LIN {X 0,Y 432.341,Z 420.255,A -85,B 0,C 180,E1 -9394.677,E2 -9394.677} C_VEL
LIN {X 0,Y 432.34,Z 420.258,A -85,B 0,C 180,E1 -9398.15,E2 -9398.15} C_VEL
LIN {X 0,Y 432.366,Z 420.256,A -85,B 0,C 180,E1 -9401.607,E2 -9401.607} C_VEL
LIN {X 0,Y 432.38,Z 420.301,A -85,B 0,C 180,E1 -9402.416,E2 -9402.416} C_VEL
LIN {X 0,Y 432.94,Z 424.326,A -85,B 0,C 180,E1 -9404.417,E2 -9404.417} C_VEL
LIN {X 0,Y 432.411,Z 431.789,A -85,B 0,C 180,E1 -9407.598,E2 -9407.598} C_VEL
LIN {X 0,Y 432.35,Z 439.582,A -85,B 0,C 180,E1 -9410.657,E2 -9410.657} C_VEL
LIN {X 0,Y 432.394,Z 447.543,A -85,B 0,C 180,E1 -9413.611,E2 -9413.611} C_VEL
LIN {X 0,Y 432.393,Z 455.479,A -85,B 0,C 180,E1 -9416.452,E2 -9416.452} C_VEL
LIN {X 0,Y 432.32,Z 464.178,A -85,B 0,C 180,E1 -9419.496,E2 -9419.496} C_VEL
LIN {X 0,Y 432.307,Z 471.048,A -85,B 0,C 180,E1 -9421.871,E2 -9421.871} C_VEL
LIN {X 0,Y 432.174,Z 480.112,A -85,B 0,C 180,E1 -9424.988,E2 -9424.988} C_VEL
LIN {X 0,Y 432.007,Z 490.424,A -85,B 0,C 180,E1 -9428.529,E2 -9428.529} C_VEL
LIN {X 0,Y 431.947,Z 493.135,A -85,B 0,C 180,E1 -9429.462,E2 -9429.462} C_VEL
LIN {X 0,Y 434.775,Z 513.471,A -85,B 0,C 180,E1 -9430.263,E2 -9430.263} C_VEL
LIN {X 0,Y 437.291,Z 527.402,A -85,B 0,C 180,E1 -9430.999,E2 -9430.999} C_VEL
LIN {X 0,Y 437.197,Z 533.625,A -85,B 0,C 180,E1 -9431.331,E2 -9431.331} C_VEL
LIN {X 0,Y 436.147,Z 551.64,A -85,B 0,C 180,E1 -9432.414,E2 -9432.414} C_VEL
LIN {X 0,Y 435.39,Z 563.892,A -85,B 0,C 180,E1 -9433.35,E2 -9433.35} C_VEL
LIN {X 0,Y 434.553,Z 575.091,A -85,B 0,C 180,E1 -9434.403,E2 -9434.403} C_VEL
LIN {X 0,Y 433.711,Z 586.298,A -85,B 0,C 180,E1 -9435.693,E2 -9435.693} C_VEL
LIN {X 0,Y 432.95,Z 596.88,A -85,B 0,C 180,E1 -9437.195,E2 -9437.195} C_VEL
LIN {X 0,Y 432.374,Z 605.824,A -85,B 0,C 180,E1 -9438.752,E2 -9438.752} C_VEL
LIN {X 0,Y 431.951,Z 612.495,A -85,B 0,C 180,E1 -9440.163,E2 -9440.163} C_VEL
LIN {X 0,Y 431.63,Z 618.023,A -85,B 0,C 180,E1 -9441.573,E2 -9441.573} C_VEL
LIN {X 0,Y 431.412,Z 623.802,A -85,B 0,C 180,E1 -9443.452,E2 -9443.452} C_VEL
LIN {X 0,Y 431.277,Z 627.993,A -85,B 0,C 180,E1 -9445.326,E2 -9445.326} C_VEL
LIN {X 0,Y 431.265,Z 630.732,A -85,B 0,C 180,E1 -9447.198,E2 -9447.198} C_VEL
LIN {X 0,Y 431.227,Z 632.093,A -85,B 0,C 180,E1 -9449.066,E2 -9449.066} C_VEL
LIN {X 0,Y 431.227,Z 632.094,A -85,B 0,C 180,E1 -9450.934,E2 -9450.934} C_VEL
LIN {X 0,Y 431.268,Z 630.735,A -85,B 0,C 180,E1 -9452.802,E2 -9452.802} C_VEL
LIN {X 0,Y 431.266,Z 627.997,A -85,B 0,C 180,E1 -9454.674,E2 -9454.674} C_VEL
LIN {X 0,Y 431.407,Z 623.802,A -85,B 0,C 180,E1 -9456.548,E2 -9456.548} C_VEL
LIN {X 0,Y 431.622,Z 618.022,A -85,B 0,C 180,E1 -9458.427,E2 -9458.427} C_VEL
LIN {X 0,Y 431.973,Z 611.488,A -85,B 0,C 180,E1 -9460.073,E2 -9460.073} C_VEL
LIN {X 0,Y 432.528,Z 603.346,A -85,B 0,C 180,E1 -9461.719,E2 -9461.719} C_VEL
LIN {X 0,Y 433.044,Z 594.648,A -85,B 0,C 180,E1 -9463.155,E2 -9463.155} C_VEL
LIN {X 0,Y 433.83,Z 584.413,A -85,B 0,C 180,E1 -9464.543,E2 -9464.543} C_VEL
LIN {X 0,Y 434.781,Z 571.943,A -85,B 0,C 180,E1 -9465.95,E2 -9465.95} C_VEL
LIN {X 0,Y 435.848,Z 559.24,A -85,B 0,C 180,E1 -9467.114,E2 -9467.114} C_VEL
LIN {X 0,Y 436.767,Z 546.427,A -85,B 0,C 180,E1 -9468.06,E2 -9468.06} C_VEL
LIN {X 0,Y 437.539,Z 533.501,A -85,B 0,C 180,E1 -9468.82,E2 -9468.82} C_VEL
LIN {X 0,Y 437.702,Z 528.722,A -85,B 0,C 180,E1 -9469.057,E2 -9469.057} C_VEL
LIN {X 0,Y 435.149,Z 514.725,A -85,B 0,C 180,E1 -9469.765,E2 -9469.765} C_VEL
LIN {X 0,Y 432.262,Z 499.953,A -85,B 0,C 180,E1 -9470.339,E2 -9470.339} C_VEL
LIN {X 0,Y 431.957,Z 497.779,A -85,B 0,C 180,E1 -9470.426,E2 -9470.426} C_VEL
LIN {X 0,Y 432.221,Z 489.918,A -85,B 0,C 180,E1 -9473.477,E2 -9473.477} C_VEL
LIN {X 0,Y 432.485,Z 481.872,A -85,B 0,C 180,E1 -9476.65,E2 -9476.65} C_VEL
LIN {X 0,Y 432.838,Z 474.315,A -85,B 0,C 180,E1 -9479.685,E2 -9479.685} C_VEL
LIN {X 0,Y 433.175,Z 466.427,A -85,B 0,C 180,E1 -9482.924,E2 -9482.924} C_VEL
LIN {X 0,Y 433.444,Z 459.515,A -85,B 0,C 180,E1 -9485.834,E2 -9485.834} C_VEL
LIN {X 0,Y 433.752,Z 451.761,A -85,B 0,C 180,E1 -9489.191,E2 -9489.191} C_VEL
LIN {X 0,Y 434.086,Z 445.759,A -85,B 0,C 180,E1 -9491.862,E2 -9491.862} C_VEL
LIN {X 0,Y 434.542,Z 438.136,A -85,B 0,C 180,E1 -9495.368,E2 -9495.368} C_VEL
LIN {X 0,Y 434.616,Z 434.256,A -85,B 0,C 180,E1 -9497.222,E2 -9497.222} C_VEL
LIN {X 0,Y 433.981,Z 429.502,A -85,B 0,C 180,E1 -9499.626,E2 -9499.626} C_VEL
LIN {X 0,Y 432.949,Z 423.719,A -85,B 0,C 180,E1 -9502.694,E2 -9502.694} C_VEL
LIN {X 0,Y 432.371,Z 420.252,A -85,B 0,C 180,E1 -9504.717,E2 -9504.717} C_VEL
LIN {X 0,Y 432.326,Z 420.259,A -85,B 0,C 180,E1 -9507.707,E2 -9507.707} C_VEL
LIN {X 0,Y 432.344,Z 420.257,A -85,B 0,C 180,E1 -9510.813,E2 -9510.813} C_VEL
LIN {X 0,Y 432.366,Z 420.243,A -85,B 0,C 180,E1 -9513.968,E2 -9513.968} C_VEL
LIN {X 0,Y 432.321,Z 420.259,A -85,B 0,C 180,E1 -9517.036,E2 -9517.036} C_VEL
LIN {X 0,Y 432.389,Z 420.245,A -85,B 0,C 180,E1 -9520.515,E2 -9520.515} C_VEL
LIN {X 0,Y 432.433,Z 420.239,A -85,B 0,C 180,E1 -9523.961,E2 -9523.961} C_VEL
LIN {X 0,Y 432.461,Z 420.242,A -85,B 0,C 180,E1 -9527.804,E2 -9527.804} C_VEL
LIN {X 0,Y 432.466,Z 420.232,A -85,B 0,C 180,E1 -9531.59,E2 -9531.59} C_VEL
LIN {X 0,Y 432.598,Z 420.224,A -85,B 0,C 180,E1 -9534.406,E2 -9534.406} C_VEL
LIN {X 0,Y 432.606,Z 420.216,A -85,B 0,C 180,E1 -9538.138,E2 -9538.138} C_VEL
LIN {X 0,Y 432.736,Z 420.21,A -85,B 0,C 180,E1 -9540,E2 -9540} C_VEL
LIN {X 0,Y 432.594,Z 420.215,A -85,B 0,C 180,E1 -9542.794,E2 -9542.794} C_VEL
LIN {X 0,Y 432.575,Z 420.226,A -85,B 0,C 180,E1 -9546.53,E2 -9546.53} C_VEL
LIN {X 0,Y 432.445,Z 420.238,A -85,B 0,C 180,E1 -9549.353,E2 -9549.353} C_VEL
LIN {X 0,Y 432.433,Z 420.241,A -85,B 0,C 180,E1 -9552.804,E2 -9552.804} C_VEL
LIN {X 0,Y 432.415,Z 420.251,A -85,B 0,C 180,E1 -9556.479,E2 -9556.479} C_VEL
LIN {X 0,Y 432.342,Z 420.257,A -85,B 0,C 180,E1 -9559.96,E2 -9559.96} C_VEL
LIN {X 0,Y 432.319,Z 420.253,A -85,B 0,C 180,E1 -9562.964,E2 -9562.964} C_VEL
LIN {X 0,Y 432.363,Z 420.25,A -85,B 0,C 180,E1 -9566.033,E2 -9566.033} C_VEL
LIN {X 0,Y 432.345,Z 420.254,A -85,B 0,C 180,E1 -9569.187,E2 -9569.187} C_VEL
LIN {X 0,Y 432.325,Z 420.258,A -85,B 0,C 180,E1 -9572.443,E2 -9572.443} C_VEL
LIN {X 0,Y 432.346,Z 420.254,A -85,B 0,C 180,E1 -9575.632,E2 -9575.632} C_VEL
LIN {X 0,Y 432.352,Z 420.256,A -85,B 0,C 180,E1 -9579.343,E2 -9579.343} C_VEL
LIN {X 0,Y 432.337,Z 420.258,A -85,B 0,C 180,E1 -9581.797,E2 -9581.797} C_VEL
LIN {X 0,Y 432.343,Z 420.256,A -85,B 0,C 180,E1 -9584.346,E2 -9584.346} C_VEL
LIN {X 0,Y 432.367,Z 420.365,A -85,B 0,C 180,E1 -9587.395,E2 -9587.395} C_VEL
LIN {X 0,Y 434.001,Z 428.984,A -85,B 0,C 180,E1 -9590.244,E2 -9590.244} C_VEL
LIN {X 0,Y 434.458,Z 432.86,A -85,B 0,C 180,E1 -9591.529,E2 -9591.529} C_VEL
LIN {X 0,Y 434.028,Z 441.711,A -85,B 0,C 180,E1 -9594.343,E2 -9594.343} C_VEL
LIN {X 0,Y 433.727,Z 452.025,A -85,B 0,C 180,E1 -9597.675,E2 -9597.675} C_VEL
LIN {X 0,Y 433.428,Z 462.73,A -85,B 0,C 180,E1 -9601.117,E2 -9601.117} C_VEL
LIN {X 0,Y 433.024,Z 473.572,A -85,B 0,C 180,E1 -9604.526,E2 -9604.526} C_VEL
LIN {X 0,Y 432.751,Z 484.213,A -85,B 0,C 180,E1 -9607.774,E2 -9607.774} C_VEL
LIN {X 0,Y 432.631,Z 491.462,A -85,B 0,C 180,E1 -9609.853,E2 -9609.853} C_VEL
LIN {X 0,Y 436.02,Z 506.623,A -85,B 0,C 180,E1 -9610.365,E2 -9610.365} C_VEL
LIN {X 0,Y 438.052,Z 518.136,A -85,B 0,C 180,E1 -9610.87,E2 -9610.87} C_VEL
LIN {X 0,Y 437.448,Z 530.781,A -85,B 0,C 180,E1 -9611.453,E2 -9611.453} C_VEL
LIN {X 0,Y 436.825,Z 543.155,A -85,B 0,C 180,E1 -9612.2,E2 -9612.2} C_VEL
LIN {X 0,Y 435.927,Z 555.472,A -85,B 0,C 180,E1 -9613.13,E2 -9613.13} C_VEL
LIN {X 0,Y 435.057,Z 566.744,A -85,B 0,C 180,E1 -9614.181,E2 -9614.181} C_VEL
LIN {X 0,Y 434.187,Z 578.069,A -85,B 0,C 180,E1 -9615.47,E2 -9615.47} C_VEL
LIN {X 0,Y 433.304,Z 588.216,A -85,B 0,C 180,E1 -9616.875,E2 -9616.875} C_VEL
LIN {X 0,Y 432.77,Z 596.592,A -85,B 0,C 180,E1 -9618.288,E2 -9618.288} C_VEL
LIN {X 0,Y 432.142,Z 604.593,A -85,B 0,C 180,E1 -9619.931,E2 -9619.931} C_VEL
LIN {X 0,Y 431.988,Z 606.62,A -85,B 0,C 180,E1 -9620.414,E2 -9620.414} C_VEL
LIN {X 0,Y 431.169,Z 609.388,A -85,B 0,C 180,E1 -9621.099,E2 -9621.099} C_VEL
LIN {X 0,Y 428.07,Z 613.464,A -85,B 0,C 180,E1 -9622.233,E2 -9622.233} C_VEL
LIN {X 0,Y 425.022,Z 616.961,A -85,B 0,C 180,E1 -9623.416,E2 -9623.416} C_VEL
LIN {X 0,Y 424.294,Z 618.757,A -85,B 0,C 180,E1 -9624.169,E2 -9624.169} C_VEL
LIN {X 0,Y 424.201,Z 620.94,A -85,B 0,C 180,E1 -9625.248,E2 -9625.248} C_VEL
LIN {X 0,Y 424.122,Z 623.658,A -85,B 0,C 180,E1 -9627.151,E2 -9627.151} C_VEL
LIN {X 0,Y 424.067,Z 625.023,A -85,B 0,C 180,E1 -9629.05,E2 -9629.05} C_VEL
LIN {X 0,Y 424.067,Z 625.061,A -85,B 0,C 180,E1 -9630.95,E2 -9630.95} C_VEL
LIN {X 0,Y 424.121,Z 623.762,A -85,B 0,C 180,E1 -9632.849,E2 -9632.849} C_VEL
LIN {X 0,Y 424.201,Z 621.106,A -85,B 0,C 180,E1 -9634.752,E2 -9634.752} C_VEL
LIN {X 0,Y 424.354,Z 617.026,A -85,B 0,C 180,E1 -9636.657,E2 -9636.657} C_VEL
LIN {X 0,Y 424.63,Z 611.396,A -85,B 0,C 180,E1 -9638.567,E2 -9638.567} C_VEL
LIN {X 0,Y 425.001,Z 606.024,A -85,B 0,C 180,E1 -9639.999,E2 -9639.999} C_VEL
LIN {X 0,Y 425.655,Z 598.336,A -85,B 0,C 180,E1 -9641.669,E2 -9641.669} C_VEL
LIN {X 0,Y 426.236,Z 590.302,A -85,B 0,C 180,E1 -9643.104,E2 -9643.104} C_VEL
LIN {X 0,Y 427.052,Z 580.624,A -85,B 0,C 180,E1 -9644.535,E2 -9644.535} C_VEL
LIN {X 0,Y 427.941,Z 569.882,A -85,B 0,C 180,E1 -9645.845,E2 -9645.845} C_VEL
LIN {X 0,Y 428.948,Z 557.958,A -85,B 0,C 180,E1 -9647.03,E2 -9647.03} C_VEL
LIN {X 0,Y 429.832,Z 546.206,A -85,B 0,C 180,E1 -9647.976,E2 -9647.976} C_VEL
LIN {X 0,Y 430.684,Z 532.74,A -85,B 0,C 180,E1 -9648.833,E2 -9648.833} C_VEL
LIN {X 0,Y 431.257,Z 518.562,A -85,B 0,C 180,E1 -9649.52,E2 -9649.52} C_VEL
LIN {X 0,Y 428.609,Z 504.1,A -85,B 0,C 180,E1 -9650.158,E2 -9650.158} C_VEL
LIN {X 0,Y 425.583,Z 491.211,A -85,B 0,C 180,E1 -9650.611,E2 -9650.611} C_VEL
LIN {X 0,Y 425.832,Z 482.093,A -85,B 0,C 180,E1 -9653.335,E2 -9653.335} C_VEL
LIN {X 0,Y 426.12,Z 472.049,A -85,B 0,C 180,E1 -9656.443,E2 -9656.443} C_VEL
LIN {X 0,Y 426.493,Z 462.064,A -85,B 0,C 180,E1 -9659.627,E2 -9659.627} C_VEL
LIN {X 0,Y 426.83,Z 451.984,A -85,B 0,C 180,E1 -9662.913,E2 -9662.913} C_VEL
LIN {X 0,Y 427.166,Z 441.511,A -85,B 0,C 180,E1 -9666.32,E2 -9666.32} C_VEL
LIN {X 0,Y 427.515,Z 434.261,A -85,B 0,C 180,E1 -9668.659,E2 -9668.659} C_VEL
LIN {X 0,Y 426.638,Z 428.084,A -85,B 0,C 180,E1 -9670.733,E2 -9670.733} C_VEL
LIN {X 0,Y 425.271,Z 421.14,A -85,B 0,C 180,E1 -9673.102,E2 -9673.102} C_VEL
LIN {X 0,Y 425.271,Z 421.14,A -85,B 0,C 180,E1 -9676.045,E2 -9676.045} C_VEL
LIN {X 0,Y 425.277,Z 421.141,A -85,B 0,C 180,E1 -9678.622,E2 -9678.622} C_VEL
LIN {X 0,Y 425.311,Z 421.136,A -85,B 0,C 180,E1 -9681.102,E2 -9681.102} C_VEL
LIN {X 0,Y 425.302,Z 421.134,A -85,B 0,C 180,E1 -9684.664,E2 -9684.664} C_VEL
LIN {X 0,Y 425.268,Z 421.138,A -85,B 0,C 180,E1 -9688.073,E2 -9688.073} C_VEL
LIN {X 0,Y 425.34,Z 421.13,A -85,B 0,C 180,E1 -9691.368,E2 -9691.368} C_VEL
LIN {X 0,Y 425.298,Z 421.133,A -85,B 0,C 180,E1 -9694.555,E2 -9694.555} C_VEL
LIN {X 0,Y 425.311,Z 421.132,A -85,B 0,C 180,E1 -9697.662,E2 -9697.662} C_VEL
LIN {X 0,Y 430.712,Z 437.499,A -85,B 0,C 180,E1 -9698.779,E2 -9698.779} C_VEL
LIN {X 0,Y 431.814,Z 441.37,A -85,B 0,C 180,E1 -9699.073,E2 -9699.073} C_VEL
LIN {X 0,Y 431.099,Z 454.659,A -85,B 0,C 180,E1 -9699.98,E2 -9699.98} C_VEL
LIN {X 0,Y 430.149,Z 467.57,A -85,B 0,C 180,E1 -9701.048,E2 -9701.048} C_VEL
LIN {X 0,Y 429.193,Z 479.566,A -85,B 0,C 180,E1 -9702.243,E2 -9702.243} C_VEL
LIN {X 0,Y 428.33,Z 490.646,A -85,B 0,C 180,E1 -9703.558,E2 -9703.558} C_VEL
LIN {X 0,Y 427.497,Z 500.849,A -85,B 0,C 180,E1 -9704.993,E2 -9704.993} C_VEL
LIN {X 0,Y 426.638,Z 510.775,A -85,B 0,C 180,E1 -9706.666,E2 -9706.666} C_VEL
LIN {X 0,Y 426.05,Z 519.022,A -85,B 0,C 180,E1 -9708.342,E2 -9708.342} C_VEL
LIN {X 0,Y 425.544,Z 525.822,A -85,B 0,C 180,E1 -9710.014,E2 -9710.014} C_VEL
LIN {X 0,Y 425.121,Z 532.087,A -85,B 0,C 180,E1 -9711.922,E2 -9711.922} C_VEL
LIN {X 0,Y 424.842,Z 536.907,A -85,B 0,C 180,E1 -9713.827,E2 -9713.827} C_VEL
LIN {X 0,Y 424.748,Z 539.643,A -85,B 0,C 180,E1 -9715.254,E2 -9715.254} C_VEL
LIN {X 0,Y 424.556,Z 542.251,A -85,B 0,C 180,E1 -9717.153,E2 -9717.153} C_VEL
LIN {X 0,Y 424.378,Z 543.678,A -85,B 0,C 180,E1 -9719.051,E2 -9719.051} C_VEL
LIN {X 0,Y 424.396,Z 543.894,A -85,B 0,C 180,E1 -9720.949,E2 -9720.949} C_VEL
LIN {X 0,Y 424.574,Z 542.936,A -85,B 0,C 180,E1 -9722.846,E2 -9722.846} C_VEL
LIN {X 0,Y 424.928,Z 540.794,A -85,B 0,C 180,E1 -9724.744,E2 -9724.744} C_VEL
LIN {X 0,Y 425.099,Z 537.458,A -85,B 0,C 180,E1 -9726.646,E2 -9726.646} C_VEL
LIN {X 0,Y 425.51,Z 532.778,A -85,B 0,C 180,E1 -9728.549,E2 -9728.549} C_VEL
LIN {X 0,Y 425.878,Z 526.647,A -85,B 0,C 180,E1 -9730.459,E2 -9730.459} C_VEL
LIN {X 0,Y 426.612,Z 518.868,A -85,B 0,C 180,E1 -9732.366,E2 -9732.366} C_VEL
LIN {X 0,Y 427.378,Z 510.571,A -85,B 0,C 180,E1 -9734.017,E2 -9734.017} C_VEL
LIN {X 0,Y 428.181,Z 501.807,A -85,B 0,C 180,E1 -9735.469,E2 -9735.469} C_VEL
LIN {X 0,Y 429.024,Z 491.512,A -85,B 0,C 180,E1 -9736.904,E2 -9736.904} C_VEL
LIN {X 0,Y 430.029,Z 479.806,A -85,B 0,C 180,E1 -9738.264,E2 -9738.264} C_VEL
LIN {X 0,Y 431.049,Z 467.92,A -85,B 0,C 180,E1 -9739.402,E2 -9739.402} C_VEL
LIN {X 0,Y 431.824,Z 456.017,A -85,B 0,C 180,E1 -9740.358,E2 -9740.358} C_VEL
LIN {X 0,Y 432.604,Z 441.693,A -85,B 0,C 180,E1 -9741.291,E2 -9741.291} C_VEL
LIN {X 0,Y 429.046,Z 430.815,A -85,B 0,C 180,E1 -9742.133,E2 -9742.133} C_VEL
LIN {X 0,Y 425.334,Z 421.52,A -85,B 0,C 180,E1 -9742.806,E2 -9742.806} C_VEL
LIN {X 0,Y 425.273,Z 421.137,A -85,B 0,C 180,E1 -9742.853,E2 -9742.853} C_VEL
LIN {X 0,Y 425.292,Z 421.139,A -85,B 0,C 180,E1 -9745.445,E2 -9745.445} C_VEL
LIN {X 0,Y 425.351,Z 421.132,A -85,B 0,C 180,E1 -9747.558,E2 -9747.558} C_VEL
LIN {X 0,Y 425.289,Z 421.133,A -85,B 0,C 180,E1 -9750.816,E2 -9750.816} C_VEL
LIN {X 0,Y 425.312,Z 421.132,A -85,B 0,C 180,E1 -9754.288,E2 -9754.288} C_VEL
LIN {X 0,Y 425.281,Z 421.138,A -85,B 0,C 180,E1 -9757.694,E2 -9757.694} C_VEL
LIN {X 0,Y 425.286,Z 421.136,A -85,B 0,C 180,E1 -9760.521,E2 -9760.521} C_VEL
LIN {X 0,Y 425.371,Z 421.276,A -85,B 0,C 180,E1 -9762.165,E2 -9762.165} C_VEL
LIN {X 0,Y 425.885,Z 424.541,A -85,B 0,C 180,E1 -9763.875,E2 -9763.875} C_VEL
LIN {X 0,Y 425.733,Z 428.375,A -85,B 0,C 180,E1 -9765.647,E2 -9765.647} C_VEL
LIN {X 0,Y 425.336,Z 438.536,A -85,B 0,C 180,E1 -9769.878,E2 -9769.878} C_VEL
LIN {X 0,Y 425.342,Z 446.633,A -85,B 0,C 180,E1 -9772.992,E2 -9772.992} C_VEL
LIN {X 0,Y 425.338,Z 454.302,A -85,B 0,C 180,E1 -9775.82,E2 -9775.82} C_VEL
LIN {X 0,Y 425.262,Z 463.858,A -85,B 0,C 180,E1 -9779.246,E2 -9779.246} C_VEL
LIN {X 0,Y 425.207,Z 471.366,A -85,B 0,C 180,E1 -9781.897,E2 -9781.897} C_VEL
LIN {X 0,Y 425.091,Z 480.314,A -85,B 0,C 180,E1 -9785.03,E2 -9785.03} C_VEL
LIN {X 0,Y 424.905,Z 490.694,A -85,B 0,C 180,E1 -9788.661,E2 -9788.661} C_VEL
LIN {X 0,Y 424.871,Z 492.011,A -85,B 0,C 180,E1 -9789.057,E2 -9789.057} C_VEL
LIN {X 0,Y 427.326,Z 508.383,A -85,B 0,C 180,E1 -9789.704,E2 -9789.704} C_VEL
LIN {X 0,Y 428.466,Z 517.12,A -85,B 0,C 180,E1 -9790.121,E2 -9790.121} C_VEL
LIN {X 0,Y 430.611,Z 530.032,A -85,B 0,C 180,E1 -9790.867,E2 -9790.867} C_VEL
LIN {X 0,Y 429.581,Z 548.076,A -85,B 0,C 180,E1 -9791.89,E2 -9791.89} C_VEL
LIN {X 0,Y 428.744,Z 560.999,A -85,B 0,C 180,E1 -9792.839,E2 -9792.839} C_VEL
LIN {X 0,Y 427.835,Z 572.697,A -85,B 0,C 180,E1 -9793.907,E2 -9793.907} C_VEL
LIN {X 0,Y 427.115,Z 582.402,A -85,B 0,C 180,E1 -9794.98,E2 -9794.98} C_VEL
LIN {X 0,Y 426.289,Z 593.119,A -85,B 0,C 180,E1 -9796.412,E2 -9796.412} C_VEL
LIN {X 0,Y 425.667,Z 601.943,A -85,B 0,C 180,E1 -9797.848,E2 -9797.848} C_VEL
LIN {X 0,Y 424.993,Z 610.376,A -85,B 0,C 180,E1 -9799.519,E2 -9799.519} C_VEL
LIN {X 0,Y 424.679,Z 616.242,A -85,B 0,C 180,E1 -9800.955,E2 -9800.955} C_VEL
LIN {X 0,Y 424.346,Z 622.488,A -85,B 0,C 180,E1 -9802.865,E2 -9802.865} C_VEL
LIN {X 0,Y 424.283,Z 626.029,A -85,B 0,C 180,E1 -9804.296,E2 -9804.296} C_VEL
LIN {X 0,Y 424.196,Z 629.481,A -85,B 0,C 180,E1 -9806.2,E2 -9806.2} C_VEL
LIN {X 0,Y 424.196,Z 631.525,A -85,B 0,C 180,E1 -9808.101,E2 -9808.101} C_VEL
LIN {X 0,Y 424.116,Z 632.205,A -85,B 0,C 180,E1 -9810,E2 -9810} C_VEL
LIN {X 0,Y 424.196,Z 631.526,A -85,B 0,C 180,E1 -9811.899,E2 -9811.899} C_VEL
LIN {X 0,Y 424.193,Z 629.485,A -85,B 0,C 180,E1 -9813.8,E2 -9813.8} C_VEL
LIN {X 0,Y 424.254,Z 626.032,A -85,B 0,C 180,E1 -9815.704,E2 -9815.704} C_VEL
LIN {X 0,Y 424.364,Z 621.062,A -85,B 0,C 180,E1 -9817.614,E2 -9817.614} C_VEL
LIN {X 0,Y 424.642,Z 616.24,A -85,B 0,C 180,E1 -9819.046,E2 -9819.046} C_VEL
LIN {X 0,Y 425.086,Z 609.261,A -85,B 0,C 180,E1 -9820.719,E2 -9820.719} C_VEL
LIN {X 0,Y 425.725,Z 600.588,A -85,B 0,C 180,E1 -9822.393,E2 -9822.393} C_VEL
LIN {X 0,Y 426.389,Z 591.492,A -85,B 0,C 180,E1 -9823.827,E2 -9823.827} C_VEL
LIN {X 0,Y 427.107,Z 582.401,A -85,B 0,C 180,E1 -9825.021,E2 -9825.021} C_VEL
LIN {X 0,Y 427.9,Z 571.524,A -85,B 0,C 180,E1 -9826.213,E2 -9826.213} C_VEL
LIN {X 0,Y 429.087,Z 557.222,A -85,B 0,C 180,E1 -9827.516,E2 -9827.516} C_VEL
LIN {X 0,Y 430.106,Z 543.368,A -85,B 0,C 180,E1 -9828.525,E2 -9828.525} C_VEL
LIN {X 0,Y 430.924,Z 530.38,A -85,B 0,C 180,E1 -9829.265,E2 -9829.265} C_VEL
LIN {X 0,Y 428.616,Z 516.863,A -85,B 0,C 180,E1 -9829.991,E2 -9829.991} C_VEL
LIN {X 0,Y 425.763,Z 501.841,A -85,B 0,C 180,E1 -9830.621,E2 -9830.621} C_VEL
LIN {X 0,Y 424.911,Z 497.198,A -85,B 0,C 180,E1 -9830.78,E2 -9830.78} C_VEL
LIN {X 0,Y 425.189,Z 489.344,A -85,B 0,C 180,E1 -9833.889,E2 -9833.889} C_VEL
LIN {X 0,Y 425.431,Z 481.945,A -85,B 0,C 180,E1 -9836.866,E2 -9836.866} C_VEL
LIN {X 0,Y 425.787,Z 475.043,A -85,B 0,C 180,E1 -9839.681,E2 -9839.681} C_VEL
LIN {X 0,Y 426.124,Z 467.15,A -85,B 0,C 180,E1 -9842.974,E2 -9842.974} C_VEL
LIN {X 0,Y 426.438,Z 459.748,A -85,B 0,C 180,E1 -9846.142,E2 -9846.142} C_VEL
LIN {X 0,Y 426.743,Z 452.616,A -85,B 0,C 180,E1 -9849.282,E2 -9849.282} C_VEL
LIN {X 0,Y 427.107,Z 446.106,A -85,B 0,C 180,E1 -9852.229,E2 -9852.229} C_VEL
LIN {X 0,Y 427.573,Z 438.808,A -85,B 0,C 180,E1 -9855.643,E2 -9855.643} C_VEL
LIN {X 0,Y 427.549,Z 434.583,A -85,B 0,C 180,E1 -9857.706,E2 -9857.706} C_VEL
LIN {X 0,Y 426.906,Z 430.032,A -85,B 0,C 180,E1 -9860.056,E2 -9860.056} C_VEL
LIN {X 0,Y 425.74,Z 423.598,A -85,B 0,C 180,E1 -9863.539,E2 -9863.539} C_VEL
LIN {X 0,Y 425.319,Z 421.13,A -85,B 0,C 180,E1 -9864.95,E2 -9864.95} C_VEL
LIN {X 0,Y 425.266,Z 421.139,A -85,B 0,C 180,E1 -9868.073,E2 -9868.073} C_VEL
LIN {X 0,Y 425.333,Z 421.133,A -85,B 0,C 180,E1 -9871.368,E2 -9871.368} C_VEL
LIN {X 0,Y 425.297,Z 421.126,A -85,B 0,C 180,E1 -9874.555,E2 -9874.555} C_VEL
LIN {X 0,Y 425.289,Z 421.132,A -85,B 0,C 180,E1 -9877.661,E2 -9877.661} C_VEL
LIN {X 0,Y 425.364,Z 421.122,A -85,B 0,C 180,E1 -9880.704,E2 -9880.704} C_VEL
LIN {X 0,Y 425.39,Z 421.117,A -85,B 0,C 180,E1 -9883.688,E2 -9883.688} C_VEL
LIN {X 0,Y 425.414,Z 421.118,A -85,B 0,C 180,E1 -9887.598,E2 -9887.598} C_VEL
LIN {X 0,Y 425.41,Z 421.109,A -85,B 0,C 180,E1 -9891.449,E2 -9891.449} C_VEL
LIN {X 0,Y 425.554,Z 421.102,A -85,B 0,C 180,E1 -9894.313,E2 -9894.313} C_VEL
LIN {X 0,Y 425.575,Z 421.091,A -85,B 0,C 180,E1 -9898.107,E2 -9898.107} C_VEL
LIN {X 0,Y 425.705,Z 421.086,A -85,B 0,C 180,E1 -9900,E2 -9900} C_VEL
LIN {X 0,Y 425.547,Z 421.092,A -85,B 0,C 180,E1 -9902.84,E2 -9902.84} C_VEL
LIN {X 0,Y 425.533,Z 421.102,A -85,B 0,C 180,E1 -9906.639,E2 -9906.639} C_VEL
LIN {X 0,Y 425.403,Z 421.117,A -85,B 0,C 180,E1 -9909.509,E2 -9909.509} C_VEL
LIN {X 0,Y 425.395,Z 421.117,A -85,B 0,C 180,E1 -9912.904,E2 -9912.904} C_VEL
LIN {X 0,Y 425.364,Z 421.128,A -85,B 0,C 180,E1 -9916.605,E2 -9916.605} C_VEL
LIN {X 0,Y 425.331,Z 421.127,A -85,B 0,C 180,E1 -9919.636,E2 -9919.636} C_VEL
LIN {X 0,Y 425.289,Z 421.132,A -85,B 0,C 180,E1 -9922.339,E2 -9922.339} C_VEL
LIN {X 0,Y 425.293,Z 421.136,A -85,B 0,C 180,E1 -9925.446,E2 -9925.446} C_VEL
LIN {X 0,Y 425.351,Z 421.127,A -85,B 0,C 180,E1 -9927.558,E2 -9927.558} C_VEL
LIN {X 0,Y 425.29,Z 421.133,A -85,B 0,C 180,E1 -9930.816,E2 -9930.816} C_VEL
LIN {X 0,Y 425.313,Z 421.133,A -85,B 0,C 180,E1 -9934.288,E2 -9934.288} C_VEL
LIN {X 0,Y 425.281,Z 421.135,A -85,B 0,C 180,E1 -9937.694,E2 -9937.694} C_VEL
LIN {X 0,Y 425.284,Z 421.138,A -85,B 0,C 180,E1 -9940.521,E2 -9940.521} C_VEL
LIN {X 0,Y 425.266,Z 421.139,A -85,B 0,C 180,E1 -9943.352,E2 -9943.352} C_VEL
LIN {X 0,Y 425.262,Z 421.142,A -85,B 0,C 180,E1 -9946.044,E2 -9946.044} C_VEL
LIN {X 0,Y 425.301,Z 421.276,A -85,B 0,C 180,E1 -9947.085,E2 -9947.085} C_VEL
LIN {X 0,Y 427.023,Z 430.139,A -85,B 0,C 180,E1 -9950.069,E2 -9950.069} C_VEL
LIN {X 0,Y 427.494,Z 435.311,A -85,B 0,C 180,E1 -9951.782,E2 -9951.782} C_VEL
LIN {X 0,Y 427.03,Z 444.714,A -85,B 0,C 180,E1 -9954.829,E2 -9954.829} C_VEL
LIN {X 0,Y 426.681,Z 455.063,A -85,B 0,C 180,E1 -9958.191,E2 -9958.191} C_VEL
LIN {X 0,Y 426.378,Z 465.095,A -85,B 0,C 180,E1 -9961.445,E2 -9961.445} C_VEL
LIN {X 0,Y 426.029,Z 475.079,A -85,B 0,C 180,E1 -9964.602,E2 -9964.602} C_VEL
LIN {X 0,Y 425.754,Z 485.137,A -85,B 0,C 180,E1 -9967.687,E2 -9967.687} C_VEL
LIN {X 0,Y 425.619,Z 491.234,A -85,B 0,C 180,E1 -9969.49,E2 -9969.49} C_VEL
LIN {X 0,Y 429.342,Z 507.939,A -85,B 0,C 180,E1 -9970.086,E2 -9970.086} C_VEL
LIN {X 0,Y 431.299,Z 519.458,A -85,B 0,C 180,E1 -9970.614,E2 -9970.614} C_VEL
LIN {X 0,Y 430.646,Z 532.803,A -85,B 0,C 180,E1 -9971.262,E2 -9971.262} C_VEL
LIN {X 0,Y 429.799,Z 546.611,A -85,B 0,C 180,E1 -9972.146,E2 -9972.146} C_VEL
LIN {X 0,Y 428.947,Z 558.279,A -85,B 0,C 180,E1 -9973.093,E2 -9973.093} C_VEL
LIN {X 0,Y 428.123,Z 567.942,A -85,B 0,C 180,E1 -9974.04,E2 -9974.04} C_VEL
LIN {X 0,Y 427.3,Z 578.124,A -85,B 0,C 180,E1 -9975.23,E2 -9975.23} C_VEL
LIN {X 0,Y 426.349,Z 588.272,A -85,B 0,C 180,E1 -9976.657,E2 -9976.657} C_VEL
LIN {X 0,Y 425.797,Z 596.649,A -85,B 0,C 180,E1 -9978.093,E2 -9978.093} C_VEL
LIN {X 0,Y 425.122,Z 604.651,A -85,B 0,C 180,E1 -9979.763,E2 -9979.763} C_VEL
LIN {X 0,Y 424.646,Z 611.088,A -85,B 0,C 180,E1 -9981.434,E2 -9981.434} C_VEL
LIN {X 0,Y 424.354,Z 616.79,A -85,B 0,C 180,E1 -9983.343,E2 -9983.343} C_VEL
LIN {X 0,Y 424.294,Z 618.757,A -85,B 0,C 180,E1 -9984.169,E2 -9984.169} C_VEL
LIN {X 0,Y 423.597,Z 620.409,A -85,B 0,C 180,E1 -9984.929,E2 -9984.929} C_VEL
LIN {X 0,Y 420.693,Z 622.599,A -85,B 0,C 180,E1 -9986.179,E2 -9986.179} C_VEL
LIN {X 0,Y 418.227,Z 623.856,A -85,B 0,C 180,E1 -9987.202,E2 -9987.202} C_VEL
LIN {X 0,Y 417.136,Z 624.512,A -85,B 0,C 180,E1 -9987.998,E2 -9987.998} C_VEL
LIN {X 0,Y 417.029,Z 624.672,A -85,B 0,C 180,E1 -9988.269,E2 -9988.269} C_VEL
LIN {X 0,Y 416.982,Z 625.267,A -85,B 0,C 180,E1 -9990,E2 -9990} C_VEL
LIN {X 0,Y 417.051,Z 624.638,A -85,B 0,C 180,E1 -9991.931,E2 -9991.931} C_VEL
LIN {X 0,Y 417.013,Z 622.664,A -85,B 0,C 180,E1 -9993.865,E2 -9993.865} C_VEL
LIN {X 0,Y 417.198,Z 619.307,A -85,B 0,C 180,E1 -9995.801,E2 -9995.801} C_VEL
LIN {X 0,Y 417.391,Z 614.471,A -85,B 0,C 180,E1 -9997.741,E2 -9997.741} C_VEL
LIN {X 0,Y 417.838,Z 608.001,A -85,B 0,C 180,E1 -9999.683,E2 -9999.683} C_VEL
LIN {X 0,Y 418.389,Z 600.791,A -85,B 0,C 180,E1 -10001.383,E2 -10001.383} C_VEL
LIN {X 0,Y 419.207,Z 592.022,A -85,B 0,C 180,E1 -10003.046,E2 -10003.046} C_VEL
LIN {X 0,Y 420.002,Z 582.419,A -85,B 0,C 180,E1 -10004.537,E2 -10004.537} C_VEL
LIN {X 0,Y 420.944,Z 572.019,A -85,B 0,C 180,E1 -10005.866,E2 -10005.866} C_VEL
LIN {X 0,Y 421.914,Z 560.542,A -85,B 0,C 180,E1 -10007.073,E2 -10007.073} C_VEL
LIN {X 0,Y 422.943,Z 547.824,A -85,B 0,C 180,E1 -10008.154,E2 -10008.154} C_VEL
LIN {X 0,Y 423.817,Z 535.216,A -85,B 0,C 180,E1 -10009.004,E2 -10009.004} C_VEL
LIN {X 0,Y 424.538,Z 521.839,A -85,B 0,C 180,E1 -10009.699,E2 -10009.699} C_VEL
LIN {X 0,Y 424.315,Z 518.305,A -85,B 0,C 180,E1 -10009.864,E2 -10009.864} C_VEL
LIN {X 0,Y 421.771,Z 504.624,A -85,B 0,C 180,E1 -10010.483,E2 -10010.483} C_VEL
LIN {X 0,Y 418.599,Z 491.165,A -85,B 0,C 180,E1 -10010.983,E2 -10010.983} C_VEL
LIN {X 0,Y 418.843,Z 482.005,A -85,B 0,C 180,E1 -10013.748,E2 -10013.748} C_VEL
LIN {X 0,Y 419.178,Z 471.873,A -85,B 0,C 180,E1 -10016.916,E2 -10016.916} C_VEL
LIN {X 0,Y 419.531,Z 461.788,A -85,B 0,C 180,E1 -10020.17,E2 -10020.17} C_VEL
LIN {X 0,Y 419.912,Z 451.597,A -85,B 0,C 180,E1 -10023.526,E2 -10023.526} C_VEL
LIN {X 0,Y 420.465,Z 439.203,A -85,B 0,C 180,E1 -10027.596,E2 -10027.596} C_VEL
LIN {X 0,Y 420.586,Z 435.52,A -85,B 0,C 180,E1 -10028.801,E2 -10028.801} C_VEL
LIN {X 0,Y 419.576,Z 428.795,A -85,B 0,C 180,E1 -10031.083,E2 -10031.083} C_VEL
LIN {X 0,Y 418.221,Z 422.016,A -85,B 0,C 180,E1 -10033.428,E2 -10033.428} C_VEL
LIN {X 0,Y 418.217,Z 422.017,A -85,B 0,C 180,E1 -10036.45,E2 -10036.45} C_VEL
LIN {X 0,Y 418.225,Z 422.021,A -85,B 0,C 180,E1 -10039.13,E2 -10039.13} C_VEL
LIN {X 0,Y 418.235,Z 422.016,A -85,B 0,C 180,E1 -10042.166,E2 -10042.166} C_VEL
LIN {X 0,Y 418.268,Z 422.006,A -85,B 0,C 180,E1 -10045.42,E2 -10045.42} C_VEL
LIN {X 0,Y 418.219,Z 422.015,A -85,B 0,C 180,E1 -10048.604,E2 -10048.604} C_VEL
LIN {X 0,Y 418.297,Z 422.006,A -85,B 0,C 180,E1 -10051.937,E2 -10051.937} C_VEL
LIN {X 0,Y 418.292,Z 422.007,A -85,B 0,C 180,E1 -10055.163,E2 -10055.163} C_VEL
LIN {X 0,Y 418.303,Z 422.191,A -85,B 0,C 180,E1 -10057.373,E2 -10057.373} C_VEL
LIN {X 0,Y 423.267,Z 437.192,A -85,B 0,C 180,E1 -10058.409,E2 -10058.409} C_VEL
LIN {X 0,Y 424.974,Z 442.506,A -85,B 0,C 180,E1 -10058.825,E2 -10058.825} C_VEL
LIN {X 0,Y 424.267,Z 455.987,A -85,B 0,C 180,E1 -10059.77,E2 -10059.77} C_VEL
LIN {X 0,Y 423.203,Z 469.96,A -85,B 0,C 180,E1 -10060.965,E2 -10060.965} C_VEL
LIN {X 0,Y 422.238,Z 481.787,A -85,B 0,C 180,E1 -10062.191,E2 -10062.191} C_VEL
LIN {X 0,Y 421.312,Z 492.639,A -85,B 0,C 180,E1 -10063.526,E2 -10063.526} C_VEL
LIN {X 0,Y 420.467,Z 502.649,A -85,B 0,C 180,E1 -10064.984,E2 -10064.984} C_VEL
LIN {X 0,Y 419.613,Z 512.413,A -85,B 0,C 180,E1 -10066.685,E2 -10066.685} C_VEL
LIN {X 0,Y 418.951,Z 520.519,A -85,B 0,C 180,E1 -10068.387,E2 -10068.387} C_VEL
LIN {X 0,Y 418.431,Z 528.044,A -85,B 0,C 180,E1 -10070.331,E2 -10070.331} C_VEL
LIN {X 0,Y 418.013,Z 533.996,A -85,B 0,C 180,E1 -10072.27,E2 -10072.27} C_VEL
LIN {X 0,Y 417.774,Z 538.542,A -85,B 0,C 180,E1 -10074.207,E2 -10074.207} C_VEL
LIN {X 0,Y 417.683,Z 541.795,A -85,B 0,C 180,E1 -10076.141,E2 -10076.141} C_VEL
LIN {X 0,Y 417.375,Z 543.865,A -85,B 0,C 180,E1 -10078.07,E2 -10078.07} C_VEL
LIN {X 0,Y 417.322,Z 544.713,A -85,B 0,C 180,E1 -10080,E2 -10080} C_VEL
LIN {X 0,Y 417.423,Z 544.373,A -85,B 0,C 180,E1 -10081.93,E2 -10081.93} C_VEL
LIN {X 0,Y 417.718,Z 542.852,A -85,B 0,C 180,E1 -10083.859,E2 -10083.859} C_VEL
LIN {X 0,Y 417.943,Z 540.149,A -85,B 0,C 180,E1 -10085.791,E2 -10085.791} C_VEL
LIN {X 0,Y 418.254,Z 536.179,A -85,B 0,C 180,E1 -10087.725,E2 -10087.725} C_VEL
LIN {X 0,Y 418.787,Z 530.818,A -85,B 0,C 180,E1 -10089.661,E2 -10089.661} C_VEL
LIN {X 0,Y 419.099,Z 525.857,A -85,B 0,C 180,E1 -10091.119,E2 -10091.119} C_VEL
LIN {X 0,Y 419.86,Z 518.741,A -85,B 0,C 180,E1 -10092.814,E2 -10092.814} C_VEL
LIN {X 0,Y 420.725,Z 510.101,A -85,B 0,C 180,E1 -10094.511,E2 -10094.511} C_VEL
LIN {X 0,Y 421.542,Z 501.239,A -85,B 0,C 180,E1 -10095.967,E2 -10095.967} C_VEL
LIN {X 0,Y 422.544,Z 490.684,A -85,B 0,C 180,E1 -10097.421,E2 -10097.421} C_VEL
LIN {X 0,Y 423.519,Z 479.255,A -85,B 0,C 180,E1 -10098.734,E2 -10098.734} C_VEL
LIN {X 0,Y 424.644,Z 466.319,A -85,B 0,C 180,E1 -10099.959,E2 -10099.959} C_VEL
LIN {X 0,Y 425.523,Z 453.93,A -85,B 0,C 180,E1 -10100.926,E2 -10100.926} C_VEL
LIN {X 0,Y 426.156,Z 443.831,A -85,B 0,C 180,E1 -10101.582,E2 -10101.582} C_VEL
LIN {X 0,Y 422.462,Z 432.497,A -85,B 0,C 180,E1 -10102.496,E2 -10102.496} C_VEL
LIN {X 0,Y 418.363,Z 422.575,A -85,B 0,C 180,E1 -10103.261,E2 -10103.261} C_VEL
LIN {X 0,Y 418.27,Z 422.01,A -85,B 0,C 180,E1 -10103.299,E2 -10103.299} C_VEL
LIN {X 0,Y 418.27,Z 422.014,A -85,B 0,C 180,E1 -10105.904,E2 -10105.904} C_VEL
LIN {X 0,Y 418.266,Z 422.012,A -85,B 0,C 180,E1 -10109.162,E2 -10109.162} C_VEL
LIN {X 0,Y 418.259,Z 422.01,A -85,B 0,C 180,E1 -10112.844,E2 -10112.844} C_VEL
LIN {X 0,Y 418.246,Z 422.013,A -85,B 0,C 180,E1 -10116.238,E2 -10116.238} C_VEL
LIN {X 0,Y 418.256,Z 422.014,A -85,B 0,C 180,E1 -10119.681,E2 -10119.681} C_VEL
LIN {X 0,Y 418.308,Z 422.131,A -85,B 0,C 180,E1 -10121.82,E2 -10121.82} C_VEL
LIN {X 0,Y 418.93,Z 425.826,A -85,B 0,C 180,E1 -10123.832,E2 -10123.832} C_VEL
LIN {X 0,Y 418.736,Z 429.868,A -85,B 0,C 180,E1 -10125.749,E2 -10125.749} C_VEL
LIN {X 0,Y 418.336,Z 439.161,A -85,B 0,C 180,E1 -10129.724,E2 -10129.724} C_VEL
LIN {X 0,Y 418.302,Z 446.892,A -85,B 0,C 180,E1 -10132.782,E2 -10132.782} C_VEL
LIN {X 0,Y 418.259,Z 455.052,A -85,B 0,C 180,E1 -10135.866,E2 -10135.866} C_VEL
LIN {X 0,Y 418.187,Z 463.578,A -85,B 0,C 180,E1 -10138.992,E2 -10138.992} C_VEL
LIN {X 0,Y 418.109,Z 471.709,A -85,B 0,C 180,E1 -10141.923,E2 -10141.923} C_VEL
LIN {X 0,Y 417.963,Z 480.967,A -85,B 0,C 180,E1 -10145.231,E2 -10145.231} C_VEL
LIN {X 0,Y 417.817,Z 490.324,A -85,B 0,C 180,E1 -10148.565,E2 -10148.565} C_VEL
LIN {X 0,Y 420.537,Z 508.269,A -85,B 0,C 180,E1 -10149.34,E2 -10149.34} C_VEL
LIN {X 0,Y 421.88,Z 519.116,A -85,B 0,C 180,E1 -10149.891,E2 -10149.891} C_VEL
LIN {X 0,Y 423.783,Z 530.959,A -85,B 0,C 180,E1 -10150.629,E2 -10150.629} C_VEL
LIN {X 0,Y 422.999,Z 546.127,A -85,B 0,C 180,E1 -10151.469,E2 -10151.469} C_VEL
LIN {X 0,Y 422.179,Z 558.027,A -85,B 0,C 180,E1 -10152.314,E2 -10152.314} C_VEL
LIN {X 0,Y 421.175,Z 570.301,A -85,B 0,C 180,E1 -10153.396,E2 -10153.396} C_VEL
LIN {X 0,Y 420.369,Z 580.378,A -85,B 0,C 180,E1 -10154.485,E2 -10154.485} C_VEL
LIN {X 0,Y 419.456,Z 591.44,A -85,B 0,C 180,E1 -10155.939,E2 -10155.939} C_VEL
LIN {X 0,Y 418.77,Z 600.536,A -85,B 0,C 180,E1 -10157.398,E2 -10157.398} C_VEL
LIN {X 0,Y 418.07,Z 609.206,A -85,B 0,C 180,E1 -10159.099,E2 -10159.099} C_VEL
LIN {X 0,Y 417.614,Z 616.186,A -85,B 0,C 180,E1 -10160.8,E2 -10160.8} C_VEL
LIN {X 0,Y 417.34,Z 621.009,A -85,B 0,C 180,E1 -10162.258,E2 -10162.258} C_VEL
LIN {X 0,Y 417.197,Z 625.972,A -85,B 0,C 180,E1 -10164.199,E2 -10164.199} C_VEL
LIN {X 0,Y 417.101,Z 629.423,A -85,B 0,C 180,E1 -10166.135,E2 -10166.135} C_VEL
LIN {X 0,Y 417.119,Z 631.467,A -85,B 0,C 180,E1 -10168.069,E2 -10168.069} C_VEL
LIN {X 0,Y 417.035,Z 632.147,A -85,B 0,C 180,E1 -10170,E2 -10170} C_VEL
LIN {X 0,Y 417.118,Z 631.468,A -85,B 0,C 180,E1 -10171.931,E2 -10171.931} C_VEL
LIN {X 0,Y 417.098,Z 629.427,A -85,B 0,C 180,E1 -10173.865,E2 -10173.865} C_VEL
LIN {X 0,Y 417.168,Z 625.975,A -85,B 0,C 180,E1 -10175.801,E2 -10175.801} C_VEL
LIN {X 0,Y 417.315,Z 621.007,A -85,B 0,C 180,E1 -10177.743,E2 -10177.743} C_VEL
LIN {X 0,Y 417.587,Z 616.185,A -85,B 0,C 180,E1 -10179.2,E2 -10179.2} C_VEL
LIN {X 0,Y 418.073,Z 609.207,A -85,B 0,C 180,E1 -10180.901,E2 -10180.901} C_VEL
LIN {X 0,Y 418.74,Z 600.535,A -85,B 0,C 180,E1 -10182.603,E2 -10182.603} C_VEL
LIN {X 0,Y 419.459,Z 591.44,A -85,B 0,C 180,E1 -10184.061,E2 -10184.061} C_VEL
LIN {X 0,Y 420.345,Z 580.375,A -85,B 0,C 180,E1 -10185.516,E2 -10185.516} C_VEL
LIN {X 0,Y 421.298,Z 569.033,A -85,B 0,C 180,E1 -10186.724,E2 -10186.724} C_VEL
LIN {X 0,Y 422.544,Z 553.658,A -85,B 0,C 180,E1 -10188.046,E2 -10188.046} C_VEL
LIN {X 0,Y 423.471,Z 541.467,A -85,B 0,C 180,E1 -10188.918,E2 -10188.918} C_VEL
LIN {X 0,Y 424.033,Z 530.278,A -85,B 0,C 180,E1 -10189.575,E2 -10189.575} C_VEL
LIN {X 0,Y 421.458,Z 515.542,A -85,B 0,C 180,E1 -10190.387,E2 -10190.387} C_VEL
LIN {X 0,Y 418.688,Z 501.063,A -85,B 0,C 180,E1 -10191.008,E2 -10191.008} C_VEL
LIN {X 0,Y 417.859,Z 496.476,A -85,B 0,C 180,E1 -10191.199,E2 -10191.199} C_VEL
LIN {X 0,Y 418.211,Z 487.466,A -85,B 0,C 180,E1 -10194.842,E2 -10194.842} C_VEL
LIN {X 0,Y 418.599,Z 478.37,A -85,B 0,C 180,E1 -10198.587,E2 -10198.587} C_VEL
LIN {X 0,Y 418.979,Z 470.501,A -85,B 0,C 180,E1 -10201.896,E2 -10201.896} C_VEL
LIN {X 0,Y 419.255,Z 463.81,A -85,B 0,C 180,E1 -10204.776,E2 -10204.776} C_VEL
LIN {X 0,Y 419.58,Z 456.35,A -85,B 0,C 180,E1 -10208.07,E2 -10208.07} C_VEL
LIN {X 0,Y 420.005,Z 449.564,A -85,B 0,C 180,E1 -10211.15,E2 -10211.15} C_VEL
LIN {X 0,Y 420.404,Z 442.221,A -85,B 0,C 180,E1 -10214.598,E2 -10214.598} C_VEL
LIN {X 0,Y 420.634,Z 437.76,A -85,B 0,C 180,E1 -10216.762,E2 -10216.762} C_VEL
LIN {X 0,Y 420.342,Z 433.751,A -85,B 0,C 180,E1 -10218.798,E2 -10218.798} C_VEL
LIN {X 0,Y 419.297,Z 427.826,A -85,B 0,C 180,E1 -10221.979,E2 -10221.979} C_VEL
LIN {X 0,Y 418.28,Z 422.007,A -85,B 0,C 180,E1 -10225.332,E2 -10225.332} C_VEL
LIN {X 0,Y 418.213,Z 422.019,A -85,B 0,C 180,E1 -10228.604,E2 -10228.604} C_VEL
LIN {X 0,Y 418.293,Z 422.005,A -85,B 0,C 180,E1 -10231.937,E2 -10231.937} C_VEL
LIN {X 0,Y 418.291,Z 422.002,A -85,B 0,C 180,E1 -10235.163,E2 -10235.163} C_VEL
LIN {X 0,Y 418.236,Z 422.009,A -85,B 0,C 180,E1 -10238.304,E2 -10238.304} C_VEL
LIN {X 0,Y 418.286,Z 422.005,A -85,B 0,C 180,E1 -10241.383,E2 -10241.383} C_VEL
LIN {X 0,Y 418.304,Z 421.998,A -85,B 0,C 180,E1 -10244.406,E2 -10244.406} C_VEL
LIN {X 0,Y 418.357,Z 421.996,A -85,B 0,C 180,E1 -10247.386,E2 -10247.386} C_VEL
LIN {X 0,Y 418.342,Z 421.992,A -85,B 0,C 180,E1 -10250.329,E2 -10250.329} C_VEL
LIN {X 0,Y 418.481,Z 421.981,A -85,B 0,C 180,E1 -10253.249,E2 -10253.249} C_VEL
LIN {X 0,Y 418.341,Z 422,A -85,B 0,C 180,E1 -10255.182,E2 -10255.182} C_VEL
LIN {X 0,Y 418.544,Z 421.966,A -85,B 0,C 180,E1 -10258.076,E2 -10258.076} C_VEL
LIN {X 0,Y 418.675,Z 421.961,A -85,B 0,C 180,E1 -10260,E2 -10260} C_VEL
LIN {X 0,Y 418.502,Z 421.969,A -85,B 0,C 180,E1 -10262.888,E2 -10262.888} C_VEL
LIN {X 0,Y 418.496,Z 421.979,A -85,B 0,C 180,E1 -10266.751,E2 -10266.751} C_VEL
LIN {X 0,Y 418.402,Z 421.982,A -85,B 0,C 180,E1 -10268.695,E2 -10268.695} C_VEL
LIN {X 0,Y 418.318,Z 422.004,A -85,B 0,C 180,E1 -10271.631,E2 -10271.631} C_VEL
LIN {X 0,Y 418.305,Z 421.998,A -85,B 0,C 180,E1 -10274.597,E2 -10274.597} C_VEL
LIN {X 0,Y 418.29,Z 422.006,A -85,B 0,C 180,E1 -10277.604,E2 -10277.604} C_VEL
LIN {X 0,Y 418.252,Z 422.012,A -85,B 0,C 180,E1 -10280.663,E2 -10280.663} C_VEL
LIN {X 0,Y 418.276,Z 422.004,A -85,B 0,C 180,E1 -10283.782,E2 -10283.782} C_VEL
LIN {X 0,Y 418.312,Z 422,A -85,B 0,C 180,E1 -10287.071,E2 -10287.071} C_VEL
LIN {X 0,Y 418.246,Z 422.009,A -85,B 0,C 180,E1 -10290.272,E2 -10290.272} C_VEL
LIN {X 0,Y 418.25,Z 422.011,A -85,B 0,C 180,E1 -10293.677,E2 -10293.677} C_VEL
LIN {X 0,Y 418.242,Z 422.014,A -85,B 0,C 180,E1 -10297.224,E2 -10297.224} C_VEL
LIN {X 0,Y 418.253,Z 422.01,A -85,B 0,C 180,E1 -10299.682,E2 -10299.682} C_VEL
LIN {X 0,Y 418.234,Z 422.017,A -85,B 0,C 180,E1 -10302.322,E2 -10302.322} C_VEL
LIN {X 0,Y 418.24,Z 422.015,A -85,B 0,C 180,E1 -10305.109,E2 -10305.109} C_VEL
LIN {X 0,Y 418.258,Z 422.211,A -85,B 0,C 180,E1 -10306.77,E2 -10306.77} C_VEL
LIN {X 0,Y 420.029,Z 431.148,A -85,B 0,C 180,E1 -10309.829,E2 -10309.829} C_VEL
LIN {X 0,Y 420.561,Z 435.179,A -85,B 0,C 180,E1 -10311.196,E2 -10311.196} C_VEL
LIN {X 0,Y 420.19,Z 443.062,A -85,B 0,C 180,E1 -10313.774,E2 -10313.774} C_VEL
LIN {X 0,Y 419.815,Z 453.511,A -85,B 0,C 180,E1 -10317.21,E2 -10317.21} C_VEL
LIN {X 0,Y 419.5,Z 463.825,A -85,B 0,C 180,E1 -10320.595,E2 -10320.595} C_VEL
LIN {X 0,Y 419.116,Z 473.247,A -85,B 0,C 180,E1 -10323.617,E2 -10323.617} C_VEL
LIN {X 0,Y 418.836,Z 483.362,A -85,B 0,C 180,E1 -10326.776,E2 -10326.776} C_VEL
LIN {X 0,Y 418.597,Z 491.28,A -85,B 0,C 180,E1 -10329.145,E2 -10329.145} C_VEL
LIN {X 0,Y 422.377,Z 507.29,A -85,B 0,C 180,E1 -10329.723,E2 -10329.723} C_VEL
LIN {X 0,Y 424.574,Z 520.457,A -85,B 0,C 180,E1 -10330.337,E2 -10330.337} C_VEL
LIN {X 0,Y 423.861,Z 533.869,A -85,B 0,C 180,E1 -10331.011,E2 -10331.011} C_VEL
LIN {X 0,Y 423.05,Z 546.657,A -85,B 0,C 180,E1 -10331.851,E2 -10331.851} C_VEL
LIN {X 0,Y 422.141,Z 558.329,A -85,B 0,C 180,E1 -10332.812,E2 -10332.812} C_VEL
LIN {X 0,Y 421.207,Z 569.128,A -85,B 0,C 180,E1 -10333.895,E2 -10333.895} C_VEL
LIN {X 0,Y 420.231,Z 580.011,A -85,B 0,C 180,E1 -10335.224,E2 -10335.224} C_VEL
LIN {X 0,Y 419.277,Z 590.438,A -85,B 0,C 180,E1 -10336.782,E2 -10336.782} C_VEL
LIN {X 0,Y 418.58,Z 599.14,A -85,B 0,C 180,E1 -10338.376,E2 -10338.376} C_VEL
LIN {X 0,Y 418.023,Z 605.7,A -85,B 0,C 180,E1 -10339.832,E2 -10339.832} C_VEL
LIN {X 0,Y 417.618,Z 611.146,A -85,B 0,C 180,E1 -10341.288,E2 -10341.288} C_VEL
LIN {X 0,Y 417.271,Z 616.849,A -85,B 0,C 180,E1 -10343.229,E2 -10343.229} C_VEL
LIN {X 0,Y 417.133,Z 620.999,A -85,B 0,C 180,E1 -10345.168,E2 -10345.168} C_VEL
LIN {X 0,Y 417.019,Z 623.717,A -85,B 0,C 180,E1 -10347.102,E2 -10347.102} C_VEL
LIN {X 0,Y 417.029,Z 624.672,A -85,B 0,C 180,E1 -10348.269,E2 -10348.269} C_VEL
LIN {X 0,Y 416.314,Z 625.107,A -85,B 0,C 180,E1 -10349.074,E2 -10349.074} C_VEL
LIN {X 0,Y 413.447,Z 625.25,A -85,B 0,C 180,E1 -10350.385,E2 -10350.385} C_VEL
LIN {X 0,Y 411.046,Z 624.951,A -85,B 0,C 180,E1 -10351.443,E2 -10351.443} C_VEL
LIN {X 0,Y 410.01,Z 624.463,A -85,B 0,C 180,E1 -10352.257,E2 -10352.257} C_VEL
LIN {X 0,Y 409.921,Z 624.224,A -85,B 0,C 180,E1 -10352.533,E2 -10352.533} C_VEL
LIN {X 0,Y 409.933,Z 622.722,A -85,B 0,C 180,E1 -10353.932,E2 -10353.932} C_VEL
LIN {X 0,Y 410.113,Z 619.364,A -85,B 0,C 180,E1 -10355.902,E2 -10355.902} C_VEL
LIN {X 0,Y 410.342,Z 614.526,A -85,B 0,C 180,E1 -10357.875,E2 -10357.875} C_VEL
LIN {X 0,Y 410.805,Z 608.056,A -85,B 0,C 180,E1 -10359.851,E2 -10359.851} C_VEL
LIN {X 0,Y 411.421,Z 600.844,A -85,B 0,C 180,E1 -10361.579,E2 -10361.579} C_VEL
LIN {X 0,Y 412.213,Z 592.378,A -85,B 0,C 180,E1 -10363.218,E2 -10363.218} C_VEL
LIN {X 0,Y 413.091,Z 582.467,A -85,B 0,C 180,E1 -10364.785,E2 -10364.785} C_VEL
LIN {X 0,Y 414.071,Z 572.064,A -85,B 0,C 180,E1 -10366.137,E2 -10366.137} C_VEL
LIN {X 0,Y 415.127,Z 560.583,A -85,B 0,C 180,E1 -10367.361,E2 -10367.361} C_VEL
LIN {X 0,Y 416.2,Z 547.859,A -85,B 0,C 180,E1 -10368.458,E2 -10368.458} C_VEL
LIN {X 0,Y 417.151,Z 534.655,A -85,B 0,C 180,E1 -10369.357,E2 -10369.357} C_VEL
LIN {X 0,Y 417.758,Z 520.411,A -85,B 0,C 180,E1 -10370.096,E2 -10370.096} C_VEL
LIN {X 0,Y 415.254,Z 506.531,A -85,B 0,C 180,E1 -10370.759,E2 -10370.759} C_VEL
LIN {X 0,Y 411.622,Z 491.159,A -85,B 0,C 180,E1 -10371.355,E2 -10371.355} C_VEL
LIN {X 0,Y 411.864,Z 481.916,A -85,B 0,C 180,E1 -10374.176,E2 -10374.176} C_VEL
LIN {X 0,Y 412.267,Z 471.695,A -85,B 0,C 180,E1 -10377.405,E2 -10377.405} C_VEL
LIN {X 0,Y 412.618,Z 461.508,A -85,B 0,C 180,E1 -10380.729,E2 -10380.729} C_VEL
LIN {X 0,Y 412.967,Z 453.175,A -85,B 0,C 180,E1 -10383.499,E2 -10383.499} C_VEL
LIN {X 0,Y 413.559,Z 440.468,A -85,B 0,C 180,E1 -10387.719,E2 -10387.719} C_VEL
LIN {X 0,Y 413.652,Z 436.765,A -85,B 0,C 180,E1 -10388.95,E2 -10388.95} C_VEL
LIN {X 0,Y 412.504,Z 429.568,A -85,B 0,C 180,E1 -10391.44,E2 -10391.44} C_VEL
LIN {X 0,Y 411.182,Z 422.893,A -85,B 0,C 180,E1 -10393.788,E2 -10393.788} C_VEL
LIN {X 0,Y 411.187,Z 422.899,A -85,B 0,C 180,E1 -10397.304,E2 -10397.304} C_VEL
LIN {X 0,Y 411.221,Z 422.889,A -85,B 0,C 180,E1 -10400.776,E2 -10400.776} C_VEL
LIN {X 0,Y 411.201,Z 422.892,A -85,B 0,C 180,E1 -10404.471,E2 -10404.471} C_VEL
LIN {X 0,Y 411.209,Z 422.887,A -85,B 0,C 180,E1 -10406.873,E2 -10406.873} C_VEL
LIN {X 0,Y 411.243,Z 422.883,A -85,B 0,C 180,E1 -10410.642,E2 -10410.642} C_VEL
LIN {X 0,Y 411.24,Z 422.886,A -85,B 0,C 180,E1 -10413.619,E2 -10413.619} C_VEL
LIN {X 0,Y 411.254,Z 422.929,A -85,B 0,C 180,E1 -10417.047,E2 -10417.047} C_VEL
LIN {X 0,Y 415.503,Z 435.81,A -85,B 0,C 180,E1 -10417.945,E2 -10417.945} C_VEL
LIN {X 0,Y 418.064,Z 443.781,A -85,B 0,C 180,E1 -10418.575,E2 -10418.575} C_VEL
LIN {X 0,Y 418.122,Z 447.907,A -85,B 0,C 180,E1 -10418.86,E2 -10418.86} C_VEL
LIN {X 0,Y 417.097,Z 461.838,A -85,B 0,C 180,E1 -10419.921,E2 -10419.921} C_VEL
LIN {X 0,Y 416.043,Z 474.374,A -85,B 0,C 180,E1 -10421.081,E2 -10421.081} C_VEL
LIN {X 0,Y 415.059,Z 486.085,A -85,B 0,C 180,E1 -10422.382,E2 -10422.382} C_VEL
LIN {X 0,Y 414.196,Z 496.41,A -85,B 0,C 180,E1 -10423.742,E2 -10423.742} C_VEL
LIN {X 0,Y 413.183,Z 507.398,A -85,B 0,C 180,E1 -10425.47,E2 -10425.47} C_VEL
LIN {X 0,Y 412.444,Z 516.492,A -85,B 0,C 180,E1 -10427.202,E2 -10427.202} C_VEL
LIN {X 0,Y 411.664,Z 524.981,A -85,B 0,C 180,E1 -10429.176,E2 -10429.176} C_VEL
LIN {X 0,Y 411.191,Z 531.762,A -85,B 0,C 180,E1 -10431.151,E2 -10431.151} C_VEL
LIN {X 0,Y 410.787,Z 537.062,A -85,B 0,C 180,E1 -10433.122,E2 -10433.122} C_VEL
LIN {X 0,Y 410.672,Z 541.002,A -85,B 0,C 180,E1 -10435.091,E2 -10435.091} C_VEL
LIN {X 0,Y 410.475,Z 543.705,A -85,B 0,C 180,E1 -10437.056,E2 -10437.056} C_VEL
LIN {X 0,Y 410.263,Z 545.202,A -85,B 0,C 180,E1 -10439.018,E2 -10439.018} C_VEL
LIN {X 0,Y 410.289,Z 545.487,A -85,B 0,C 180,E1 -10440.981,E2 -10440.981} C_VEL
LIN {X 0,Y 410.492,Z 544.593,A -85,B 0,C 180,E1 -10442.944,E2 -10442.944} C_VEL
LIN {X 0,Y 410.895,Z 542.508,A -85,B 0,C 180,E1 -10444.906,E2 -10444.906} C_VEL
LIN {X 0,Y 411.099,Z 539.231,A -85,B 0,C 180,E1 -10446.873,E2 -10446.873} C_VEL
LIN {X 0,Y 411.601,Z 534.603,A -85,B 0,C 180,E1 -10448.84,E2 -10448.84} C_VEL
LIN {X 0,Y 412.023,Z 528.533,A -85,B 0,C 180,E1 -10450.814,E2 -10450.814} C_VEL
LIN {X 0,Y 412.863,Z 520.8,A -85,B 0,C 180,E1 -10452.785,E2 -10452.785} C_VEL
LIN {X 0,Y 413.746,Z 512.587,A -85,B 0,C 180,E1 -10454.484,E2 -10454.484} C_VEL
LIN {X 0,Y 414.656,Z 503.861,A -85,B 0,C 180,E1 -10455.987,E2 -10455.987} C_VEL
LIN {X 0,Y 415.613,Z 493.648,A -85,B 0,C 180,E1 -10457.467,E2 -10457.467} C_VEL
LIN {X 0,Y 416.764,Z 482.009,A -85,B 0,C 180,E1 -10458.871,E2 -10458.871} C_VEL
LIN {X 0,Y 417.963,Z 468.946,A -85,B 0,C 180,E1 -10460.164,E2 -10460.164} C_VEL
LIN {X 0,Y 418.878,Z 456.904,A -85,B 0,C 180,E1 -10461.145,E2 -10461.145} C_VEL
LIN {X 0,Y 419.578,Z 445.35,A -85,B 0,C 180,E1 -10461.938,E2 -10461.938} C_VEL
LIN {X 0,Y 415.94,Z 434.406,A -85,B 0,C 180,E1 -10462.869,E2 -10462.869} C_VEL
LIN {X 0,Y 411.33,Z 423.429,A -85,B 0,C 180,E1 -10463.769,E2 -10463.769} C_VEL
LIN {X 0,Y 411.257,Z 422.885,A -85,B 0,C 180,E1 -10463.833,E2 -10463.833} C_VEL
LIN {X 0,Y 411.26,Z 422.887,A -85,B 0,C 180,E1 -10467.478,E2 -10467.478} C_VEL
LIN {X 0,Y 411.191,Z 422.89,A -85,B 0,C 180,E1 -10470.847,E2 -10470.847} C_VEL
LIN {X 0,Y 411.207,Z 422.889,A -85,B 0,C 180,E1 -10474.333,E2 -10474.333} C_VEL
LIN {X 0,Y 411.197,Z 422.892,A -85,B 0,C 180,E1 -10477.973,E2 -10477.973} C_VEL
LIN {X 0,Y 411.259,Z 423.029,A -85,B 0,C 180,E1 -10481.473,E2 -10481.473} C_VEL
LIN {X 0,Y 411.928,Z 426.815,A -85,B 0,C 180,E1 -10483.63,E2 -10483.63} C_VEL
LIN {X 0,Y 411.771,Z 430.813,A -85,B 0,C 180,E1 -10485.591,E2 -10485.591} C_VEL
LIN {X 0,Y 411.32,Z 439.684,A -85,B 0,C 180,E1 -10489.512,E2 -10489.512} C_VEL
LIN {X 0,Y 411.241,Z 447.392,A -85,B 0,C 180,E1 -10492.65,E2 -10492.65} C_VEL
LIN {X 0,Y 411.203,Z 455.171,A -85,B 0,C 180,E1 -10495.666,E2 -10495.666} C_VEL
LIN {X 0,Y 411.14,Z 463.314,A -85,B 0,C 180,E1 -10498.726,E2 -10498.726} C_VEL
LIN {X 0,Y 411.021,Z 472.068,A -85,B 0,C 180,E1 -10501.951,E2 -10501.951} C_VEL
LIN {X 0,Y 410.858,Z 481.52,A -85,B 0,C 180,E1 -10505.395,E2 -10505.395} C_VEL
LIN {X 0,Y 410.739,Z 488.84,A -85,B 0,C 180,E1 -10508.052,E2 -10508.052} C_VEL
LIN {X 0,Y 413.707,Z 507.072,A -85,B 0,C 180,E1 -10508.902,E2 -10508.902} C_VEL
LIN {X 0,Y 415.211,Z 520.592,A -85,B 0,C 180,E1 -10509.631,E2 -10509.631} C_VEL
LIN {X 0,Y 416.975,Z 531.762,A -85,B 0,C 180,E1 -10510.356,E2 -10510.356} C_VEL
LIN {X 0,Y 416.313,Z 545.069,A -85,B 0,C 180,E1 -10511.094,E2 -10511.094} C_VEL
LIN {X 0,Y 415.389,Z 557.988,A -85,B 0,C 180,E1 -10512.015,E2 -10512.015} C_VEL
LIN {X 0,Y 414.353,Z 570.256,A -85,B 0,C 180,E1 -10513.114,E2 -10513.114} C_VEL
LIN {X 0,Y 413.506,Z 580.33,A -85,B 0,C 180,E1 -10514.22,E2 -10514.22} C_VEL
LIN {X 0,Y 412.518,Z 591.389,A -85,B 0,C 180,E1 -10515.698,E2 -10515.698} C_VEL
LIN {X 0,Y 411.797,Z 600.483,A -85,B 0,C 180,E1 -10517.181,E2 -10517.181} C_VEL
LIN {X 0,Y 411.043,Z 609.152,A -85,B 0,C 180,E1 -10518.91,E2 -10518.91} C_VEL
LIN {X 0,Y 410.569,Z 616.131,A -85,B 0,C 180,E1 -10520.641,E2 -10520.641} C_VEL
LIN {X 0,Y 410.275,Z 620.952,A -85,B 0,C 180,E1 -10522.123,E2 -10522.123} C_VEL
LIN {X 0,Y 410.117,Z 625.915,A -85,B 0,C 180,E1 -10524.098,E2 -10524.098} C_VEL
LIN {X 0,Y 410.012,Z 629.365,A -85,B 0,C 180,E1 -10526.068,E2 -10526.068} C_VEL
LIN {X 0,Y 410.043,Z 631.409,A -85,B 0,C 180,E1 -10528.036,E2 -10528.036} C_VEL
LIN {X 0,Y 409.955,Z 632.088,A -85,B 0,C 180,E1 -10530,E2 -10530} C_VEL
LIN {X 0,Y 410.042,Z 631.41,A -85,B 0,C 180,E1 -10531.964,E2 -10531.964} C_VEL
LIN {X 0,Y 410.007,Z 629.369,A -85,B 0,C 180,E1 -10533.932,E2 -10533.932} C_VEL
LIN {X 0,Y 410.085,Z 625.918,A -85,B 0,C 180,E1 -10535.902,E2 -10535.902} C_VEL
LIN {X 0,Y 410.257,Z 620.95,A -85,B 0,C 180,E1 -10537.877,E2 -10537.877} C_VEL
LIN {X 0,Y 410.549,Z 616.129,A -85,B 0,C 180,E1 -10539.359,E2 -10539.359} C_VEL
LIN {X 0,Y 411.04,Z 609.152,A -85,B 0,C 180,E1 -10541.09,E2 -10541.09} C_VEL
LIN {X 0,Y 411.743,Z 600.481,A -85,B 0,C 180,E1 -10542.82,E2 -10542.82} C_VEL
LIN {X 0,Y 412.521,Z 591.387,A -85,B 0,C 180,E1 -10544.302,E2 -10544.302} C_VEL
LIN {X 0,Y 413.471,Z 580.324,A -85,B 0,C 180,E1 -10545.781,E2 -10545.781} C_VEL
LIN {X 0,Y 414.468,Z 568.985,A -85,B 0,C 180,E1 -10547.008,E2 -10547.008} C_VEL
LIN {X 0,Y 415.492,Z 556.404,A -85,B 0,C 180,E1 -10548.108,E2 -10548.108} C_VEL
LIN {X 0,Y 416.789,Z 540.04,A -85,B 0,C 180,E1 -10549.293,E2 -10549.293} C_VEL
LIN {X 0,Y 417.19,Z 531.2,A -85,B 0,C 180,E1 -10549.827,E2 -10549.827} C_VEL
LIN {X 0,Y 414.698,Z 516.344,A -85,B 0,C 180,E1 -10550.689,E2 -10550.689} C_VEL
LIN {X 0,Y 412.006,Z 501.946,A -85,B 0,C 180,E1 -10551.34,E2 -10551.34} C_VEL
LIN {X 0,Y 410.817,Z 495.869,A -85,B 0,C 180,E1 -10551.58,E2 -10551.58} C_VEL
LIN {X 0,Y 411.181,Z 486.854,A -85,B 0,C 180,E1 -10555.297,E2 -10555.297} C_VEL
LIN {X 0,Y 411.589,Z 478.001,A -85,B 0,C 180,E1 -10559.01,E2 -10559.01} C_VEL
LIN {X 0,Y 411.967,Z 469.856,A -85,B 0,C 180,E1 -10562.505,E2 -10562.505} C_VEL
LIN {X 0,Y 412.263,Z 463.219,A -85,B 0,C 180,E1 -10565.423,E2 -10565.423} C_VEL
LIN {X 0,Y 412.573,Z 456.587,A -85,B 0,C 180,E1 -10568.409,E2 -10568.409} C_VEL
LIN {X 0,Y 413.024,Z 449.734,A -85,B 0,C 180,E1 -10571.577,E2 -10571.577} C_VEL
LIN {X 0,Y 413.563,Z 441.469,A -85,B 0,C 180,E1 -10575.54,E2 -10575.54} C_VEL
LIN {X 0,Y 413.576,Z 436.887,A -85,B 0,C 180,E1 -10577.838,E2 -10577.838} C_VEL
LIN {X 0,Y 413.016,Z 432.851,A -85,B 0,C 180,E1 -10579.972,E2 -10579.972} C_VEL
LIN {X 0,Y 411.878,Z 426.777,A -85,B 0,C 180,E1 -10583.329,E2 -10583.329} C_VEL
LIN {X 0,Y 411.215,Z 422.888,A -85,B 0,C 180,E1 -10585.667,E2 -10585.667} C_VEL
LIN {X 0,Y 411.191,Z 422.892,A -85,B 0,C 180,E1 -10589.153,E2 -10589.153} C_VEL
LIN {X 0,Y 411.26,Z 422.882,A -85,B 0,C 180,E1 -10592.522,E2 -10592.522} C_VEL
LIN {X 0,Y 411.229,Z 422.885,A -85,B 0,C 180,E1 -10595.785,E2 -10595.785} C_VEL
LIN {X 0,Y 411.198,Z 422.879,A -85,B 0,C 180,E1 -10598.966,E2 -10598.966} C_VEL
LIN {X 0,Y 411.255,Z 422.885,A -85,B 0,C 180,E1 -10602.085,E2 -10602.085} C_VEL
LIN {X 0,Y 411.262,Z 422.87,A -85,B 0,C 180,E1 -10605.147,E2 -10605.147} C_VEL
LIN {X 0,Y 411.286,Z 422.88,A -85,B 0,C 180,E1 -10608.167,E2 -10608.167} C_VEL
LIN {X 0,Y 411.44,Z 422.851,A -85,B 0,C 180,E1 -10612.191,E2 -10612.191} C_VEL
LIN {X 0,Y 411.473,Z 422.857,A -85,B 0,C 180,E1 -10614.118,E2 -10614.118} C_VEL
LIN {X 0,Y 411.513,Z 422.842,A -85,B 0,C 180,E1 -10618.043,E2 -10618.043} C_VEL
LIN {X 0,Y 411.644,Z 422.837,A -85,B 0,C 180,E1 -10620,E2 -10620} C_VEL
LIN {X 0,Y 411.459,Z 422.846,A -85,B 0,C 180,E1 -10622.937,E2 -10622.937} C_VEL
LIN {X 0,Y 411.463,Z 422.855,A -85,B 0,C 180,E1 -10626.867,E2 -10626.867} C_VEL
LIN {X 0,Y 411.356,Z 422.859,A -85,B 0,C 180,E1 -10628.845,E2 -10628.845} C_VEL
LIN {X 0,Y 411.286,Z 422.881,A -85,B 0,C 180,E1 -10631.833,E2 -10631.833} C_VEL
LIN {X 0,Y 411.262,Z 422.877,A -85,B 0,C 180,E1 -10634.853,E2 -10634.853} C_VEL
LIN {X 0,Y 411.255,Z 422.878,A -85,B 0,C 180,E1 -10637.915,E2 -10637.915} C_VEL
LIN {X 0,Y 411.199,Z 422.893,A -85,B 0,C 180,E1 -10641.034,E2 -10641.034} C_VEL
LIN {X 0,Y 411.221,Z 422.887,A -85,B 0,C 180,E1 -10644.216,E2 -10644.216} C_VEL
LIN {X 0,Y 411.261,Z 422.881,A -85,B 0,C 180,E1 -10647.478,E2 -10647.478} C_VEL
LIN {X 0,Y 411.191,Z 422.89,A -85,B 0,C 180,E1 -10650.848,E2 -10650.848} C_VEL
LIN {X 0,Y 411.207,Z 422.89,A -85,B 0,C 180,E1 -10654.334,E2 -10654.334} C_VEL
LIN {X 0,Y 411.197,Z 422.89,A -85,B 0,C 180,E1 -10657.974,E2 -10657.974} C_VEL
LIN {X 0,Y 411.184,Z 422.894,A -85,B 0,C 180,E1 -10660.504,E2 -10660.504} C_VEL
LIN {X 0,Y 411.18,Z 422.893,A -85,B 0,C 180,E1 -10663.133,E2 -10663.133} C_VEL
LIN {X 0,Y 411.212,Z 423.077,A -85,B 0,C 180,E1 -10666.413,E2 -10666.413} C_VEL
LIN {X 0,Y 412.792,Z 430.911,A -85,B 0,C 180,E1 -10669.138,E2 -10669.138} C_VEL
LIN {X 0,Y 413.629,Z 436.423,A -85,B 0,C 180,E1 -10671.048,E2 -10671.048} C_VEL
LIN {X 0,Y 413.305,Z 443.769,A -85,B 0,C 180,E1 -10673.476,E2 -10673.476} C_VEL
LIN {X 0,Y 412.875,Z 454.352,A -85,B 0,C 180,E1 -10676.995,E2 -10676.995} C_VEL
LIN {X 0,Y 412.547,Z 464.614,A -85,B 0,C 180,E1 -10680.394,E2 -10680.394} C_VEL
LIN {X 0,Y 412.123,Z 474.785,A -85,B 0,C 180,E1 -10683.68,E2 -10683.68} C_VEL
LIN {X 0,Y 411.789,Z 485.924,A -85,B 0,C 180,E1 -10687.164,E2 -10687.164} C_VEL
LIN {X 0,Y 411.644,Z 491.227,A -85,B 0,C 180,E1 -10688.76,E2 -10688.76} C_VEL
LIN {X 0,Y 415.621,Z 508.212,A -85,B 0,C 180,E1 -10689.407,E2 -10689.407} C_VEL
LIN {X 0,Y 417.849,Z 521.443,A -85,B 0,C 180,E1 -10690.05,E2 -10690.05} C_VEL
LIN {X 0,Y 417.107,Z 534.599,A -85,B 0,C 180,E1 -10690.732,E2 -10690.732} C_VEL
LIN {X 0,Y 416.166,Z 548.256,A -85,B 0,C 180,E1 -10691.668,E2 -10691.668} C_VEL
LIN {X 0,Y 415.09,Z 560.906,A -85,B 0,C 180,E1 -10692.765,E2 -10692.765} C_VEL
LIN {X 0,Y 414.036,Z 572.328,A -85,B 0,C 180,E1 -10693.988,E2 -10693.988} C_VEL
LIN {X 0,Y 412.983,Z 583.561,A -85,B 0,C 180,E1 -10695.463,E2 -10695.463} C_VEL
LIN {X 0,Y 412.26,Z 591.84,A -85,B 0,C 180,E1 -10696.785,E2 -10696.785} C_VEL
LIN {X 0,Y 411.456,Z 600.409,A -85,B 0,C 180,E1 -10698.422,E2 -10698.422} C_VEL
LIN {X 0,Y 410.83,Z 607.719,A -85,B 0,C 180,E1 -10700.15,E2 -10700.15} C_VEL
LIN {X 0,Y 410.345,Z 614.26,A -85,B 0,C 180,E1 -10702.125,E2 -10702.125} C_VEL
LIN {X 0,Y 410.123,Z 619.168,A -85,B 0,C 180,E1 -10704.099,E2 -10704.099} C_VEL
LIN {X 0,Y 409.933,Z 622.59,A -85,B 0,C 180,E1 -10706.068,E2 -10706.068} C_VEL
LIN {X 0,Y 409.962,Z 624.624,A -85,B 0,C 180,E1 -10708.035,E2 -10708.035} C_VEL
LIN {X 0,Y 409.905,Z 625.326,A -85,B 0,C 180,E1 -10710,E2 -10710} C_VEL
LIN {X 0,Y 409.961,Z 624.696,A -85,B 0,C 180,E1 -10711.965,E2 -10711.965} C_VEL
LIN {X 0,Y 409.921,Z 624.224,A -85,B 0,C 180,E1 -10712.533,E2 -10712.533} C_VEL
LIN {X 0,Y 409.246,Z 623.455,A -85,B 0,C 180,E1 -10713.346,E2 -10713.346} C_VEL
LIN {X 0,Y 406.428,Z 621.751,A -85,B 0,C 180,E1 -10714.66,E2 -10714.66} C_VEL
LIN {X 0,Y 404.095,Z 619.996,A -85,B 0,C 180,E1 -10715.709,E2 -10715.709} C_VEL
LIN {X 0,Y 403.149,Z 618.368,A -85,B 0,C 180,E1 -10716.508,E2 -10716.508} C_VEL
LIN {X 0,Y 403.102,Z 617.726,A -85,B 0,C 180,E1 -10716.777,E2 -10716.777} C_VEL
LIN {X 0,Y 403.404,Z 613.151,A -85,B 0,C 180,E1 -10718.516,E2 -10718.516} C_VEL
LIN {X 0,Y 403.786,Z 608.111,A -85,B 0,C 180,E1 -10720.024,E2 -10720.024} C_VEL
LIN {X 0,Y 404.451,Z 600.897,A -85,B 0,C 180,E1 -10721.781,E2 -10721.781} C_VEL
LIN {X 0,Y 405.224,Z 592.948,A -85,B 0,C 180,E1 -10723.357,E2 -10723.357} C_VEL
LIN {X 0,Y 406.024,Z 584.241,A -85,B 0,C 180,E1 -10724.792,E2 -10724.792} C_VEL
LIN {X 0,Y 407.055,Z 574.198,A -85,B 0,C 180,E1 -10726.165,E2 -10726.165} C_VEL
LIN {X 0,Y 408.084,Z 563.145,A -85,B 0,C 180,E1 -10727.411,E2 -10727.411} C_VEL
LIN {X 0,Y 409.239,Z 550.967,A -85,B 0,C 180,E1 -10728.524,E2 -10728.524} C_VEL
LIN {X 0,Y 410.168,Z 538.793,A -85,B 0,C 180,E1 -10729.422,E2 -10729.422} C_VEL
LIN {X 0,Y 411.035,Z 524.506,A -85,B 0,C 180,E1 -10730.238,E2 -10730.238} C_VEL
LIN {X 0,Y 411.141,Z 522.19,A -85,B 0,C 180,E1 -10730.353,E2 -10730.353} C_VEL
LIN {X 0,Y 408.672,Z 508.119,A -85,B 0,C 180,E1 -10731.059,E2 -10731.059} C_VEL
LIN {X 0,Y 405.166,Z 493.414,A -85,B 0,C 180,E1 -10731.635,E2 -10731.635} C_VEL
LIN {X 0,Y 404.631,Z 491.154,A -85,B 0,C 180,E1 -10731.743,E2 -10731.743} C_VEL
LIN {X 0,Y 404.902,Z 481.825,A -85,B 0,C 180,E1 -10734.619,E2 -10734.619} C_VEL
LIN {X 0,Y 405.34,Z 471.514,A -85,B 0,C 180,E1 -10737.914,E2 -10737.914} C_VEL
LIN {X 0,Y 405.718,Z 461.222,A -85,B 0,C 180,E1 -10741.31,E2 -10741.31} C_VEL
LIN {X 0,Y 406.148,Z 450.796,A -85,B 0,C 180,E1 -10744.822,E2 -10744.822} C_VEL
LIN {X 0,Y 406.729,Z 439.919,A -85,B 0,C 180,E1 -10748.466,E2 -10748.466} C_VEL
LIN {X 0,Y 406.457,Z 436.121,A -85,B 0,C 180,E1 -10749.774,E2 -10749.774} C_VEL
LIN {X 0,Y 405.013,Z 428.104,A -85,B 0,C 180,E1 -10752.59,E2 -10752.59} C_VEL
LIN {X 0,Y 404.123,Z 423.774,A -85,B 0,C 180,E1 -10754.189,E2 -10754.189} C_VEL
LIN {X 0,Y 404.142,Z 423.777,A -85,B 0,C 180,E1 -10757.296,E2 -10757.296} C_VEL
LIN {X 0,Y 404.17,Z 423.77,A -85,B 0,C 180,E1 -10759.955,E2 -10759.955} C_VEL
LIN {X 0,Y 404.141,Z 423.766,A -85,B 0,C 180,E1 -10763.124,E2 -10763.124} C_VEL
LIN {X 0,Y 404.147,Z 423.761,A -85,B 0,C 180,E1 -10766.188,E2 -10766.188} C_VEL
LIN {X 0,Y 404.155,Z 423.758,A -85,B 0,C 180,E1 -10769.716,E2 -10769.716} C_VEL
LIN {X 0,Y 404.197,Z 423.762,A -85,B 0,C 180,E1 -10773.123,E2 -10773.123} C_VEL
LIN {X 0,Y 404.181,Z 423.764,A -85,B 0,C 180,E1 -10776.426,E2 -10776.426} C_VEL
LIN {X 0,Y 404.174,Z 423.764,A -85,B 0,C 180,E1 -10776.724,E2 -10776.724} C_VEL
LIN {X 0,Y 409.116,Z 438.66,A -85,B 0,C 180,E1 -10777.795,E2 -10777.795} C_VEL
LIN {X 0,Y 411.448,Z 446.452,A -85,B 0,C 180,E1 -10778.426,E2 -10778.426} C_VEL
LIN {X 0,Y 410.498,Z 460.164,A -85,B 0,C 180,E1 -10779.453,E2 -10779.453} C_VEL
LIN {X 0,Y 409.359,Z 473.807,A -85,B 0,C 180,E1 -10780.702,E2 -10780.702} C_VEL
LIN {X 0,Y 408.266,Z 486.19,A -85,B 0,C 180,E1 -10782.079,E2 -10782.079} C_VEL
LIN {X 0,Y 407.193,Z 498.306,A -85,B 0,C 180,E1 -10783.712,E2 -10783.712} C_VEL
LIN {X 0,Y 406.29,Z 507.713,A -85,B 0,C 180,E1 -10785.218,E2 -10785.218} C_VEL
LIN {X 0,Y 405.593,Z 515.717,A -85,B 0,C 180,E1 -10786.739,E2 -10786.739} C_VEL
LIN {X 0,Y 404.868,Z 523.478,A -85,B 0,C 180,E1 -10788.485,E2 -10788.485} C_VEL
LIN {X 0,Y 404.311,Z 530.752,A -85,B 0,C 180,E1 -10790.495,E2 -10790.495} C_VEL
LIN {X 0,Y 403.891,Z 536.918,A -85,B 0,C 180,E1 -10792.677,E2 -10792.677} C_VEL
LIN {X 0,Y 403.675,Z 539.846,A -85,B 0,C 180,E1 -10794.004,E2 -10794.004} C_VEL
LIN {X 0,Y 403.618,Z 543.197,A -85,B 0,C 180,E1 -10796.006,E2 -10796.006} C_VEL
LIN {X 0,Y 403.274,Z 545.348,A -85,B 0,C 180,E1 -10798.002,E2 -10798.002} C_VEL
LIN {X 0,Y 403.209,Z 546.271,A -85,B 0,C 180,E1 -10800,E2 -10800} C_VEL
LIN {X 0,Y 403.326,Z 546.013,A -85,B 0,C 180,E1 -10801.997,E2 -10801.997} C_VEL
LIN {X 0,Y 403.669,Z 544.564,A -85,B 0,C 180,E1 -10803.993,E2 -10803.993} C_VEL
LIN {X 0,Y 403.928,Z 541.932,A -85,B 0,C 180,E1 -10805.992,E2 -10805.992} C_VEL
LIN {X 0,Y 404.325,Z 538.017,A -85,B 0,C 180,E1 -10807.993,E2 -10807.993} C_VEL
LIN {X 0,Y 404.909,Z 532.723,A -85,B 0,C 180,E1 -10809.995,E2 -10809.995} C_VEL
LIN {X 0,Y 405.291,Z 527.817,A -85,B 0,C 180,E1 -10811.503,E2 -10811.503} C_VEL
LIN {X 0,Y 406.149,Z 520.767,A -85,B 0,C 180,E1 -10813.255,E2 -10813.255} C_VEL
LIN {X 0,Y 407.132,Z 512.2,A -85,B 0,C 180,E1 -10815.007,E2 -10815.007} C_VEL
LIN {X 0,Y 408.075,Z 503.427,A -85,B 0,C 180,E1 -10816.509,E2 -10816.509} C_VEL
LIN {X 0,Y 409.23,Z 492.979,A -85,B 0,C 180,E1 -10818.007,E2 -10818.007} C_VEL
LIN {X 0,Y 410.185,Z 483.136,A -85,B 0,C 180,E1 -10819.198,E2 -10819.198} C_VEL
LIN {X 0,Y 411.436,Z 470.305,A -85,B 0,C 180,E1 -10820.498,E2 -10820.498} C_VEL
LIN {X 0,Y 412.407,Z 458.457,A -85,B 0,C 180,E1 -10821.493,E2 -10821.493} C_VEL
LIN {X 0,Y 413.202,Z 447.564,A -85,B 0,C 180,E1 -10822.259,E2 -10822.259} C_VEL
LIN {X 0,Y 409.493,Z 436.538,A -85,B 0,C 180,E1 -10823.25,E2 -10823.25} C_VEL
LIN {X 0,Y 405.048,Z 426.385,A -85,B 0,C 180,E1 -10824.147,E2 -10824.147} C_VEL
LIN {X 0,Y 404.183,Z 423.768,A -85,B 0,C 180,E1 -10824.367,E2 -10824.367} C_VEL
LIN {X 0,Y 404.197,Z 423.766,A -85,B 0,C 180,E1 -10828,E2 -10828} C_VEL
LIN {X 0,Y 404.141,Z 423.771,A -85,B 0,C 180,E1 -10831.558,E2 -10831.558} C_VEL
LIN {X 0,Y 404.186,Z 423.764,A -85,B 0,C 180,E1 -10835.016,E2 -10835.016} C_VEL
LIN {X 0,Y 404.158,Z 423.768,A -85,B 0,C 180,E1 -10838.757,E2 -10838.757} C_VEL
LIN {X 0,Y 404.178,Z 423.811,A -85,B 0,C 180,E1 -10841.026,E2 -10841.026} C_VEL
LIN {X 0,Y 404.831,Z 427.411,A -85,B 0,C 180,E1 -10843.186,E2 -10843.186} C_VEL
LIN {X 0,Y 404.964,Z 430.15,A -85,B 0,C 180,E1 -10844.64,E2 -10844.64} C_VEL
LIN {X 0,Y 404.29,Z 438.155,A -85,B 0,C 180,E1 -10848.374,E2 -10848.374} C_VEL
LIN {X 0,Y 404.233,Z 445.394,A -85,B 0,C 180,E1 -10851.478,E2 -10851.478} C_VEL
LIN {X 0,Y 404.198,Z 454.098,A -85,B 0,C 180,E1 -10854.985,E2 -10854.985} C_VEL
LIN {X 0,Y 404.052,Z 463.328,A -85,B 0,C 180,E1 -10858.546,E2 -10858.546} C_VEL
LIN {X 0,Y 403.991,Z 470.943,A -85,B 0,C 180,E1 -10861.419,E2 -10861.419} C_VEL
LIN {X 0,Y 403.792,Z 480.108,A -85,B 0,C 180,E1 -10864.831,E2 -10864.831} C_VEL
LIN {X 0,Y 403.664,Z 487.365,A -85,B 0,C 180,E1 -10867.519,E2 -10867.519} C_VEL
LIN {X 0,Y 404.367,Z 491.188,A -85,B 0,C 180,E1 -10867.701,E2 -10867.701} C_VEL
LIN {X 0,Y 406.785,Z 505.272,A -85,B 0,C 180,E1 -10868.4,E2 -10868.4} C_VEL
LIN {X 0,Y 408.362,Z 520.722,A -85,B 0,C 180,E1 -10869.27,E2 -10869.27} C_VEL
LIN {X 0,Y 410.266,Z 532.983,A -85,B 0,C 180,E1 -10870.084,E2 -10870.084} C_VEL
LIN {X 0,Y 409.503,Z 546.813,A -85,B 0,C 180,E1 -10870.885,E2 -10870.885} C_VEL
LIN {X 0,Y 408.525,Z 559.452,A -85,B 0,C 180,E1 -10871.832,E2 -10871.832} C_VEL
LIN {X 0,Y 407.406,Z 571.387,A -85,B 0,C 180,E1 -10872.947,E2 -10872.947} C_VEL
LIN {X 0,Y 406.465,Z 582.255,A -85,B 0,C 180,E1 -10874.197,E2 -10874.197} C_VEL
LIN {X 0,Y 405.469,Z 592.965,A -85,B 0,C 180,E1 -10875.7,E2 -10875.7} C_VEL
LIN {X 0,Y 404.724,Z 601.784,A -85,B 0,C 180,E1 -10877.209,E2 -10877.209} C_VEL
LIN {X 0,Y 404.045,Z 609.098,A -85,B 0,C 180,E1 -10878.715,E2 -10878.715} C_VEL
LIN {X 0,Y 403.539,Z 616.076,A -85,B 0,C 180,E1 -10880.477,E2 -10880.477} C_VEL
LIN {X 0,Y 403.134,Z 622.318,A -85,B 0,C 180,E1 -10882.487,E2 -10882.487} C_VEL
LIN {X 0,Y 403.045,Z 625.858,A -85,B 0,C 180,E1 -10883.995,E2 -10883.995} C_VEL
LIN {X 0,Y 402.926,Z 629.308,A -85,B 0,C 180,E1 -10885.999,E2 -10885.999} C_VEL
LIN {X 0,Y 402.95,Z 631.35,A -85,B 0,C 180,E1 -10888.001,E2 -10888.001} C_VEL
LIN {X 0,Y 402.879,Z 632.03,A -85,B 0,C 180,E1 -10890,E2 -10890} C_VEL
LIN {X 0,Y 402.95,Z 631.352,A -85,B 0,C 180,E1 -10891.999,E2 -10891.999} C_VEL
LIN {X 0,Y 402.919,Z 629.311,A -85,B 0,C 180,E1 -10894.001,E2 -10894.001} C_VEL
LIN {X 0,Y 402.994,Z 625.86,A -85,B 0,C 180,E1 -10896.006,E2 -10896.006} C_VEL
LIN {X 0,Y 403.194,Z 620.893,A -85,B 0,C 180,E1 -10898.016,E2 -10898.016} C_VEL
LIN {X 0,Y 403.523,Z 616.073,A -85,B 0,C 180,E1 -10899.524,E2 -10899.524} C_VEL
LIN {X 0,Y 404.033,Z 609.095,A -85,B 0,C 180,E1 -10901.285,E2 -10901.285} C_VEL
LIN {X 0,Y 404.68,Z 601.779,A -85,B 0,C 180,E1 -10902.793,E2 -10902.793} C_VEL
LIN {X 0,Y 405.469,Z 592.959,A -85,B 0,C 180,E1 -10904.3,E2 -10904.3} C_VEL
LIN {X 0,Y 406.434,Z 582.246,A -85,B 0,C 180,E1 -10905.804,E2 -10905.804} C_VEL
LIN {X 0,Y 407.406,Z 571.376,A -85,B 0,C 180,E1 -10907.053,E2 -10907.053} C_VEL
LIN {X 0,Y 408.478,Z 559.441,A -85,B 0,C 180,E1 -10908.171,E2 -10908.171} C_VEL
LIN {X 0,Y 409.505,Z 546.499,A -85,B 0,C 180,E1 -10909.135,E2 -10909.135} C_VEL
LIN {X 0,Y 410.457,Z 532.973,A -85,B 0,C 180,E1 -10910.026,E2 -10910.026} C_VEL
LIN {X 0,Y 408.082,Z 518.256,A -85,B 0,C 180,E1 -10910.926,E2 -10910.926} C_VEL
LIN {X 0,Y 405.411,Z 503.483,A -85,B 0,C 180,E1 -10911.642,E2 -10911.642} C_VEL
LIN {X 0,Y 403.755,Z 495.232,A -85,B 0,C 180,E1 -10911.978,E2 -10911.978} C_VEL
LIN {X 0,Y 404.102,Z 487.407,A -85,B 0,C 180,E1 -10915.262,E2 -10915.262} C_VEL
LIN {X 0,Y 404.532,Z 478.406,A -85,B 0,C 180,E1 -10919.107,E2 -10919.107} C_VEL
LIN {X 0,Y 404.922,Z 470.519,A -85,B 0,C 180,E1 -10922.551,E2 -10922.551} C_VEL
LIN {X 0,Y 405.216,Z 464.153,A -85,B 0,C 180,E1 -10925.397,E2 -10925.397} C_VEL
LIN {X 0,Y 405.588,Z 456.806,A -85,B 0,C 180,E1 -10928.762,E2 -10928.762} C_VEL
LIN {X 0,Y 406.021,Z 450.139,A -85,B 0,C 180,E1 -10931.9,E2 -10931.9} C_VEL
LIN {X 0,Y 406.567,Z 442.343,A -85,B 0,C 180,E1 -10935.697,E2 -10935.697} C_VEL
LIN {X 0,Y 406.56,Z 437.796,A -85,B 0,C 180,E1 -10938.015,E2 -10938.015} C_VEL
LIN {X 0,Y 405.985,Z 433.782,A -85,B 0,C 180,E1 -10940.17,E2 -10940.17} C_VEL
LIN {X 0,Y 405.067,Z 428.832,A -85,B 0,C 180,E1 -10942.95,E2 -10942.95} C_VEL
LIN {X 0,Y 404.159,Z 423.766,A -85,B 0,C 180,E1 -10945.964,E2 -10945.964} C_VEL
LIN {X 0,Y 404.147,Z 423.771,A -85,B 0,C 180,E1 -10949.715,E2 -10949.715} C_VEL
LIN {X 0,Y 404.196,Z 423.753,A -85,B 0,C 180,E1 -10953.123,E2 -10953.123} C_VEL
LIN {X 0,Y 404.179,Z 423.76,A -85,B 0,C 180,E1 -10955.335,E2 -10955.335} C_VEL
LIN {X 0,Y 404.141,Z 423.761,A -85,B 0,C 180,E1 -10958.581,E2 -10958.581} C_VEL
LIN {X 0,Y 404.212,Z 423.76,A -85,B 0,C 180,E1 -10961.762,E2 -10961.762} C_VEL
LIN {X 0,Y 404.208,Z 423.748,A -85,B 0,C 180,E1 -10964.882,E2 -10964.882} C_VEL
LIN {X 0,Y 404.258,Z 423.757,A -85,B 0,C 180,E1 -10967.959,E2 -10967.959} C_VEL
LIN {X 0,Y 404.268,Z 423.74,A -85,B 0,C 180,E1 -10970.999,E2 -10970.999} C_VEL
LIN {X 0,Y 404.42,Z 423.737,A -85,B 0,C 180,E1 -10974.015,E2 -10974.015} C_VEL
LIN {X 0,Y 404.482,Z 423.717,A -85,B 0,C 180,E1 -10978.009,E2 -10978.009} C_VEL
LIN {X 0,Y 404.614,Z 423.713,A -85,B 0,C 180,E1 -10980,E2 -10980} C_VEL
LIN {X 0,Y 404.417,Z 423.722,A -85,B 0,C 180,E1 -10982.989,E2 -10982.989} C_VEL
LIN {X 0,Y 404.414,Z 423.733,A -85,B 0,C 180,E1 -10986.987,E2 -10986.987} C_VEL
LIN {X 0,Y 404.261,Z 423.75,A -85,B 0,C 180,E1 -10990.012,E2 -10990.012} C_VEL
LIN {X 0,Y 404.268,Z 423.747,A -85,B 0,C 180,E1 -10993.211,E2 -10993.211} C_VEL
LIN {X 0,Y 404.218,Z 423.759,A -85,B 0,C 180,E1 -10997.007,E2 -10997.007} C_VEL
LIN {X 0,Y 404.166,Z 423.766,A -85,B 0,C 180,E1 -11000.352,E2 -11000.352} C_VEL
LIN {X 0,Y 404.165,Z 423.761,A -85,B 0,C 180,E1 -11003.575,E2 -11003.575} C_VEL
LIN {X 0,Y 404.185,Z 423.761,A -85,B 0,C 180,E1 -11005.766,E2 -11005.766} C_VEL
LIN {X 0,Y 404.197,Z 423.761,A -85,B 0,C 180,E1 -11008,E2 -11008} C_VEL
LIN {X 0,Y 404.141,Z 423.772,A -85,B 0,C 180,E1 -11011.558,E2 -11011.558} C_VEL
LIN {X 0,Y 404.186,Z 423.762,A -85,B 0,C 180,E1 -11015.016,E2 -11015.016} C_VEL
LIN {X 0,Y 404.157,Z 423.769,A -85,B 0,C 180,E1 -11018.757,E2 -11018.757} C_VEL
LIN {X 0,Y 404.126,Z 423.772,A -85,B 0,C 180,E1 -11021.6,E2 -11021.6} C_VEL
LIN {X 0,Y 404.151,Z 423.768,A -85,B 0,C 180,E1 -11024.523,E2 -11024.523} C_VEL
LIN {X 0,Y 404.158,Z 423.868,A -85,B 0,C 180,E1 -11026.015,E2 -11026.015} C_VEL
LIN {X 0,Y 406.006,Z 433.116,A -85,B 0,C 180,E1 -11029.284,E2 -11029.284} C_VEL
LIN {X 0,Y 406.733,Z 438.142,A -85,B 0,C 180,E1 -11031.038,E2 -11031.038} C_VEL
LIN {X 0,Y 406.311,Z 446.895,A -85,B 0,C 180,E1 -11033.978,E2 -11033.978} C_VEL
LIN {X 0,Y 405.862,Z 457.468,A -85,B 0,C 180,E1 -11037.534,E2 -11037.534} C_VEL
LIN {X 0,Y 405.502,Z 467.8,A -85,B 0,C 180,E1 -11040.969,E2 -11040.969} C_VEL
LIN {X 0,Y 405.053,Z 478.55,A -85,B 0,C 180,E1 -11044.455,E2 -11044.455} C_VEL
LIN {X 0,Y 404.731,Z 488.457,A -85,B 0,C 180,E1 -11047.541,E2 -11047.541} C_VEL
LIN {X 0,Y 404.679,Z 491.223,A -85,B 0,C 180,E1 -11048.376,E2 -11048.376} C_VEL
LIN {X 0,Y 408.629,Z 508.024,A -85,B 0,C 180,E1 -11049.032,E2 -11049.032} C_VEL
LIN {X 0,Y 410.973,Z 521.21,A -85,B 0,C 180,E1 -11049.69,E2 -11049.69} C_VEL
LIN {X 0,Y 410.86,Z 527.263,A -85,B 0,C 180,E1 -11049.994,E2 -11049.994} C_VEL
LIN {X 0,Y 410.069,Z 540.211,A -85,B 0,C 180,E1 -11050.765,E2 -11050.765} C_VEL
LIN {X 0,Y 409.111,Z 552.887,A -85,B 0,C 180,E1 -11051.729,E2 -11051.729} C_VEL
LIN {X 0,Y 407.877,Z 564.659,A -85,B 0,C 180,E1 -11052.838,E2 -11052.838} C_VEL
LIN {X 0,Y 406.986,Z 574.459,A -85,B 0,C 180,E1 -11053.961,E2 -11053.961} C_VEL
LIN {X 0,Y 405.92,Z 585.249,A -85,B 0,C 180,E1 -11055.46,E2 -11055.46} C_VEL
LIN {X 0,Y 405.272,Z 592.446,A -85,B 0,C 180,E1 -11056.649,E2 -11056.649} C_VEL
LIN {X 0,Y 404.492,Z 600.467,A -85,B 0,C 180,E1 -11058.22,E2 -11058.22} C_VEL
LIN {X 0,Y 403.815,Z 607.778,A -85,B 0,C 180,E1 -11059.977,E2 -11059.977} C_VEL
LIN {X 0,Y 403.29,Z 614.318,A -85,B 0,C 180,E1 -11061.986,E2 -11061.986} C_VEL
LIN {X 0,Y 403.066,Z 619.227,A -85,B 0,C 180,E1 -11063.995,E2 -11063.995} C_VEL
LIN {X 0,Y 402.855,Z 622.649,A -85,B 0,C 180,E1 -11065.999,E2 -11065.999} C_VEL
LIN {X 0,Y 402.859,Z 624.683,A -85,B 0,C 180,E1 -11068.001,E2 -11068.001} C_VEL
LIN {X 0,Y 402.831,Z 625.384,A -85,B 0,C 180,E1 -11070,E2 -11070} C_VEL
LIN {X 0,Y 402.858,Z 624.754,A -85,B 0,C 180,E1 -11071.999,E2 -11071.999} C_VEL
LIN {X 0,Y 402.855,Z 622.779,A -85,B 0,C 180,E1 -11074.001,E2 -11074.001} C_VEL
LIN {X 0,Y 403.024,Z 619.421,A -85,B 0,C 180,E1 -11076.006,E2 -11076.006} C_VEL
LIN {X 0,Y 403.102,Z 617.726,A -85,B 0,C 180,E1 -11076.777,E2 -11076.777} C_VEL
LIN {X 0,Y 402.556,Z 615.859,A -85,B 0,C 180,E1 -11077.569,E2 -11077.569} C_VEL
LIN {X 0,Y 399.944,Z 612.423,A -85,B 0,C 180,E1 -11078.846,E2 -11078.846} C_VEL
LIN {X 0,Y 397.392,Z 608.465,A -85,B 0,C 180,E1 -11080.103,E2 -11080.103} C_VEL
LIN {X 0,Y 396.951,Z 605.686,A -85,B 0,C 180,E1 -11080.857,E2 -11080.857} C_VEL
LIN {X 0,Y 397.739,Z 598.547,A -85,B 0,C 180,E1 -11082.501,E2 -11082.501} C_VEL
LIN {X 0,Y 398.519,Z 590.227,A -85,B 0,C 180,E1 -11084.083,E2 -11084.083} C_VEL
LIN {X 0,Y 399.51,Z 580.816,A -85,B 0,C 180,E1 -11085.561,E2 -11085.561} C_VEL
LIN {X 0,Y 400.627,Z 570.06,A -85,B 0,C 180,E1 -11086.956,E2 -11086.956} C_VEL
LIN {X 0,Y 401.811,Z 558.113,A -85,B 0,C 180,E1 -11088.219,E2 -11088.219} C_VEL
LIN {X 0,Y 402.888,Z 546.332,A -85,B 0,C 180,E1 -11089.224,E2 -11089.224} C_VEL
LIN {X 0,Y 403.851,Z 533.63,A -85,B 0,C 180,E1 -11090.088,E2 -11090.088} C_VEL
LIN {X 0,Y 404.358,Z 522.885,A -85,B 0,C 180,E1 -11090.674,E2 -11090.674} C_VEL
LIN {X 0,Y 401.947,Z 509.03,A -85,B 0,C 180,E1 -11091.399,E2 -11091.399} C_VEL
LIN {X 0,Y 398.564,Z 494.848,A -85,B 0,C 180,E1 -11091.982,E2 -11091.982} C_VEL
LIN {X 0,Y 397.7,Z 491.204,A -85,B 0,C 180,E1 -11092.125,E2 -11092.125} C_VEL
LIN {X 0,Y 398.043,Z 480.595,A -85,B 0,C 180,E1 -11095.435,E2 -11095.435} C_VEL
LIN {X 0,Y 398.419,Z 471.328,A -85,B 0,C 180,E1 -11098.442,E2 -11098.442} C_VEL
LIN {X 0,Y 398.817,Z 460.928,A -85,B 0,C 180,E1 -11101.915,E2 -11101.915} C_VEL
LIN {X 0,Y 399.211,Z 452.155,A -85,B 0,C 180,E1 -11104.901,E2 -11104.901} C_VEL
LIN {X 0,Y 399.834,Z 441.25,A -85,B 0,C 180,E1 -11108.608,E2 -11108.608} C_VEL
LIN {X 0,Y 399.512,Z 437.406,A -85,B 0,C 180,E1 -11109.947,E2 -11109.947} C_VEL
LIN {X 0,Y 398.027,Z 429.229,A -85,B 0,C 180,E1 -11112.881,E2 -11112.881} C_VEL
LIN {X 0,Y 397.123,Z 424.644,A -85,B 0,C 180,E1 -11114.579,E2 -11114.579} C_VEL
LIN {X 0,Y 397.07,Z 424.655,A -85,B 0,C 180,E1 -11118.021,E2 -11118.021} C_VEL
LIN {X 0,Y 397.133,Z 424.645,A -85,B 0,C 180,E1 -11121.138,E2 -11121.138} C_VEL
LIN {X 0,Y 397.122,Z 424.645,A -85,B 0,C 180,E1 -11124.496,E2 -11124.496} C_VEL
LIN {X 0,Y 397.083,Z 424.65,A -85,B 0,C 180,E1 -11127.929,E2 -11127.929} C_VEL
LIN {X 0,Y 397.129,Z 424.644,A -85,B 0,C 180,E1 -11131.457,E2 -11131.457} C_VEL
LIN {X 0,Y 397.155,Z 424.639,A -85,B 0,C 180,E1 -11134.487,E2 -11134.487} C_VEL
LIN {X 0,Y 397.166,Z 424.745,A -85,B 0,C 180,E1 -11136.407,E2 -11136.407} C_VEL
LIN {X 0,Y 402.059,Z 439.604,A -85,B 0,C 180,E1 -11137.5,E2 -11137.5} C_VEL
LIN {X 0,Y 404.651,Z 448.313,A -85,B 0,C 180,E1 -11138.221,E2 -11138.221} C_VEL
LIN {X 0,Y 403.542,Z 462.792,A -85,B 0,C 180,E1 -11139.349,E2 -11139.349} C_VEL
LIN {X 0,Y 402.357,Z 476.055,A -85,B 0,C 180,E1 -11140.617,E2 -11140.617} C_VEL
LIN {X 0,Y 401.364,Z 487.203,A -85,B 0,C 180,E1 -11141.892,E2 -11141.892} C_VEL
LIN {X 0,Y 400.347,Z 498.455,A -85,B 0,C 180,E1 -11143.425,E2 -11143.425} C_VEL
LIN {X 0,Y 399.396,Z 507.936,A -85,B 0,C 180,E1 -11144.957,E2 -11144.957} C_VEL
LIN {X 0,Y 398.643,Z 516.136,A -85,B 0,C 180,E1 -11146.526,E2 -11146.526} C_VEL
LIN {X 0,Y 397.885,Z 523.88,A -85,B 0,C 180,E1 -11148.28,E2 -11148.28} C_VEL
LIN {X 0,Y 397.322,Z 531.235,A -85,B 0,C 180,E1 -11150.326,E2 -11150.326} C_VEL
LIN {X 0,Y 396.871,Z 537.028,A -85,B 0,C 180,E1 -11152.368,E2 -11152.368} C_VEL
LIN {X 0,Y 396.624,Z 540.474,A -85,B 0,C 180,E1 -11153.897,E2 -11153.897} C_VEL
LIN {X 0,Y 396.587,Z 543.884,A -85,B 0,C 180,E1 -11155.935,E2 -11155.935} C_VEL
LIN {X 0,Y 396.227,Z 546.08,A -85,B 0,C 180,E1 -11157.967,E2 -11157.967} C_VEL
LIN {X 0,Y 396.153,Z 547.055,A -85,B 0,C 180,E1 -11160,E2 -11160} C_VEL
LIN {X 0,Y 396.279,Z 546.843,A -85,B 0,C 180,E1 -11162.033,E2 -11162.033} C_VEL
LIN {X 0,Y 396.647,Z 545.431,A -85,B 0,C 180,E1 -11164.064,E2 -11164.064} C_VEL
LIN {X 0,Y 396.924,Z 542.845,A -85,B 0,C 180,E1 -11166.098,E2 -11166.098} C_VEL
LIN {X 0,Y 397.366,Z 538.984,A -85,B 0,C 180,E1 -11168.134,E2 -11168.134} C_VEL
LIN {X 0,Y 397.978,Z 533.727,A -85,B 0,C 180,E1 -11170.171,E2 -11170.171} C_VEL
LIN {X 0,Y 398.401,Z 528.836,A -85,B 0,C 180,E1 -11171.705,E2 -11171.705} C_VEL
LIN {X 0,Y 399.328,Z 521.835,A -85,B 0,C 180,E1 -11173.485,E2 -11173.485} C_VEL
LIN {X 0,Y 400.393,Z 513.353,A -85,B 0,C 180,E1 -11175.265,E2 -11175.265} C_VEL
LIN {X 0,Y 401.383,Z 504.609,A -85,B 0,C 180,E1 -11176.792,E2 -11176.792} C_VEL
LIN {X 0,Y 402.587,Z 494.231,A -85,B 0,C 180,E1 -11178.314,E2 -11178.314} C_VEL
LIN {X 0,Y 403.64,Z 484.374,A -85,B 0,C 180,E1 -11179.539,E2 -11179.539} C_VEL
LIN {X 0,Y 404.937,Z 471.797,A -85,B 0,C 180,E1 -11180.842,E2 -11180.842} C_VEL
LIN {X 0,Y 406.096,Z 458.47,A -85,B 0,C 180,E1 -11181.978,E2 -11181.978} C_VEL
LIN {X 0,Y 406.777,Z 449.458,A -85,B 0,C 180,E1 -11182.63,E2 -11182.63} C_VEL
LIN {X 0,Y 403.145,Z 438.736,A -85,B 0,C 180,E1 -11183.638,E2 -11183.638} C_VEL
LIN {X 0,Y 398.194,Z 427.565,A -85,B 0,C 180,E1 -11184.698,E2 -11184.698} C_VEL
LIN {X 0,Y 397.167,Z 424.641,A -85,B 0,C 180,E1 -11184.962,E2 -11184.962} C_VEL
LIN {X 0,Y 397.163,Z 424.643,A -85,B 0,C 180,E1 -11187.776,E2 -11187.776} C_VEL
LIN {X 0,Y 397.08,Z 424.648,A -85,B 0,C 180,E1 -11190.882,E2 -11190.882} C_VEL
LIN {X 0,Y 397.126,Z 424.643,A -85,B 0,C 180,E1 -11194.493,E2 -11194.493} C_VEL
LIN {X 0,Y 397.105,Z 424.647,A -85,B 0,C 180,E1 -11198.275,E2 -11198.275} C_VEL
LIN {X 0,Y 397.152,Z 424.719,A -85,B 0,C 180,E1 -11200.631,E2 -11200.631} C_VEL
LIN {X 0,Y 397.96,Z 429.576,A -85,B 0,C 180,E1 -11203.609,E2 -11203.609} C_VEL
LIN {X 0,Y 397.745,Z 433.694,A -85,B 0,C 180,E1 -11205.737,E2 -11205.737} C_VEL
LIN {X 0,Y 397.252,Z 442.883,A -85,B 0,C 180,E1 -11209.984,E2 -11209.984} C_VEL
LIN {X 0,Y 397.134,Z 451.528,A -85,B 0,C 180,E1 -11213.641,E2 -11213.641} C_VEL
LIN {X 0,Y 397.037,Z 459.183,A -85,B 0,C 180,E1 -11216.72,E2 -11216.72} C_VEL
LIN {X 0,Y 396.903,Z 466.783,A -85,B 0,C 180,E1 -11219.685,E2 -11219.685} C_VEL
LIN {X 0,Y 396.832,Z 474.342,A -85,B 0,C 180,E1 -11222.583,E2 -11222.583} C_VEL
LIN {X 0,Y 396.667,Z 483.228,A -85,B 0,C 180,E1 -11225.952,E2 -11225.952} C_VEL
LIN {X 0,Y 396.608,Z 485.82,A -85,B 0,C 180,E1 -11226.931,E2 -11226.931} C_VEL
LIN {X 0,Y 397.289,Z 489.557,A -85,B 0,C 180,E1 -11227.117,E2 -11227.117} C_VEL
LIN {X 0,Y 399.762,Z 502.646,A -85,B 0,C 180,E1 -11227.815,E2 -11227.815} C_VEL
LIN {X 0,Y 401.225,Z 516.517,A -85,B 0,C 180,E1 -11228.611,E2 -11228.611} C_VEL
LIN {X 0,Y 402.375,Z 526.589,A -85,B 0,C 180,E1 -11229.294,E2 -11229.294} C_VEL
LIN {X 0,Y 403.528,Z 534.347,A -85,B 0,C 180,E1 -11229.809,E2 -11229.809} C_VEL
LIN {X 0,Y 402.681,Z 547.94,A -85,B 0,C 180,E1 -11230.634,E2 -11230.634} C_VEL
LIN {X 0,Y 401.609,Z 560.835,A -85,B 0,C 180,E1 -11231.64,E2 -11231.64} C_VEL
LIN {X 0,Y 400.481,Z 572.514,A -85,B 0,C 180,E1 -11232.774,E2 -11232.774} C_VEL
LIN {X 0,Y 399.595,Z 582.207,A -85,B 0,C 180,E1 -11233.918,E2 -11233.918} C_VEL
LIN {X 0,Y 398.544,Z 592.914,A -85,B 0,C 180,E1 -11235.446,E2 -11235.446} C_VEL
LIN {X 0,Y 397.747,Z 601.731,A -85,B 0,C 180,E1 -11236.98,E2 -11236.98} C_VEL
LIN {X 0,Y 397.059,Z 609.043,A -85,B 0,C 180,E1 -11238.514,E2 -11238.514} C_VEL
LIN {X 0,Y 396.492,Z 616.02,A -85,B 0,C 180,E1 -11240.306,E2 -11240.306} C_VEL
LIN {X 0,Y 396.159,Z 620.84,A -85,B 0,C 180,E1 -11241.841,E2 -11241.841} C_VEL
LIN {X 0,Y 395.977,Z 625.801,A -85,B 0,C 180,E1 -11243.887,E2 -11243.887} C_VEL
LIN {X 0,Y 395.842,Z 629.25,A -85,B 0,C 180,E1 -11245.928,E2 -11245.928} C_VEL
LIN {X 0,Y 395.844,Z 631.292,A -85,B 0,C 180,E1 -11247.965,E2 -11247.965} C_VEL
LIN {X 0,Y 395.805,Z 631.971,A -85,B 0,C 180,E1 -11250,E2 -11250} C_VEL
LIN {X 0,Y 395.844,Z 631.293,A -85,B 0,C 180,E1 -11252.035,E2 -11252.035} C_VEL
LIN {X 0,Y 395.834,Z 629.253,A -85,B 0,C 180,E1 -11254.073,E2 -11254.073} C_VEL
LIN {X 0,Y 395.909,Z 625.802,A -85,B 0,C 180,E1 -11256.114,E2 -11256.114} C_VEL
LIN {X 0,Y 396.148,Z 620.835,A -85,B 0,C 180,E1 -11258.159,E2 -11258.159} C_VEL
LIN {X 0,Y 396.626,Z 614.206,A -85,B 0,C 180,E1 -11260.206,E2 -11260.206} C_VEL
LIN {X 0,Y 397.26,Z 606.782,A -85,B 0,C 180,E1 -11261.998,E2 -11261.998} C_VEL
LIN {X 0,Y 397.948,Z 598.746,A -85,B 0,C 180,E1 -11263.578,E2 -11263.578} C_VEL
LIN {X 0,Y 398.85,Z 589.597,A -85,B 0,C 180,E1 -11265.064,E2 -11265.064} C_VEL
LIN {X 0,Y 399.837,Z 579.154,A -85,B 0,C 180,E1 -11266.465,E2 -11266.465} C_VEL
LIN {X 0,Y 400.987,Z 567.598,A -85,B 0,C 180,E1 -11267.73,E2 -11267.73} C_VEL
LIN {X 0,Y 402.141,Z 554.737,A -85,B 0,C 180,E1 -11268.864,E2 -11268.864} C_VEL
LIN {X 0,Y 403.07,Z 542.088,A -85,B 0,C 180,E1 -11269.744,E2 -11269.744} C_VEL
LIN {X 0,Y 403.535,Z 533.276,A -85,B 0,C 180,E1 -11270.318,E2 -11270.318} C_VEL
LIN {X 0,Y 401.385,Z 519.617,A -85,B 0,C 180,E1 -11271.193,E2 -11271.193} C_VEL
LIN {X 0,Y 398.778,Z 504.904,A -85,B 0,C 180,E1 -11271.948,E2 -11271.948} C_VEL
LIN {X 0,Y 396.703,Z 494.569,A -85,B 0,C 180,E1 -11272.389,E2 -11272.389} C_VEL
LIN {X 0,Y 397.05,Z 487.351,A -85,B 0,C 180,E1 -11275.481,E2 -11275.481} C_VEL
LIN {X 0,Y 397.469,Z 479.048,A -85,B 0,C 180,E1 -11279.095,E2 -11279.095} C_VEL
LIN {X 0,Y 397.862,Z 471.162,A -85,B 0,C 180,E1 -11282.6,E2 -11282.6} C_VEL
LIN {X 0,Y 398.192,Z 464.303,A -85,B 0,C 180,E1 -11285.719,E2 -11285.719} C_VEL
LIN {X 0,Y 398.616,Z 457,A -85,B 0,C 180,E1 -11289.126,E2 -11289.126} C_VEL
LIN {X 0,Y 399.055,Z 450.396,A -85,B 0,C 180,E1 -11292.295,E2 -11292.295} C_VEL
LIN {X 0,Y 399.491,Z 444.365,A -85,B 0,C 180,E1 -11295.276,E2 -11295.276} C_VEL
LIN {X 0,Y 399.608,Z 439.792,A -85,B 0,C 180,E1 -11297.618,E2 -11297.618} C_VEL
LIN {X 0,Y 399.051,Z 435.385,A -85,B 0,C 180,E1 -11299.997,E2 -11299.997} C_VEL
LIN {X 0,Y 398.039,Z 429.922,A -85,B 0,C 180,E1 -11303.107,E2 -11303.107} C_VEL
LIN {X 0,Y 397.122,Z 424.643,A -85,B 0,C 180,E1 -11306.282,E2 -11306.282} C_VEL
LIN {X 0,Y 397.106,Z 424.649,A -85,B 0,C 180,E1 -11310.135,E2 -11310.135} C_VEL
LIN {X 0,Y 397.196,Z 424.631,A -85,B 0,C 180,E1 -11312.61,E2 -11312.61} C_VEL
LIN {X 0,Y 397.134,Z 424.642,A -85,B 0,C 180,E1 -11315.982,E2 -11315.982} C_VEL
LIN {X 0,Y 397.14,Z 424.628,A -85,B 0,C 180,E1 -11319.705,E2 -11319.705} C_VEL
LIN {X 0,Y 397.183,Z 424.635,A -85,B 0,C 180,E1 -11322.845,E2 -11322.845} C_VEL
LIN {X 0,Y 397.23,Z 424.626,A -85,B 0,C 180,E1 -11326.703,E2 -11326.703} C_VEL
LIN {X 0,Y 397.219,Z 424.624,A -85,B 0,C 180,E1 -11329.809,E2 -11329.809} C_VEL
LIN {X 0,Y 397.34,Z 424.615,A -85,B 0,C 180,E1 -11332.888,E2 -11332.888} C_VEL
LIN {X 0,Y 397.256,Z 424.626,A -85,B 0,C 180,E1 -11334.925,E2 -11334.925} C_VEL
LIN {X 0,Y 397.451,Z 424.592,A -85,B 0,C 180,E1 -11337.973,E2 -11337.973} C_VEL
LIN {X 0,Y 397.583,Z 424.589,A -85,B 0,C 180,E1 -11340,E2 -11340} C_VEL
LIN {X 0,Y 397.377,Z 424.599,A -85,B 0,C 180,E1 -11343.042,E2 -11343.042} C_VEL
LIN {X 0,Y 397.366,Z 424.611,A -85,B 0,C 180,E1 -11347.112,E2 -11347.112} C_VEL
LIN {X 0,Y 397.22,Z 424.628,A -85,B 0,C 180,E1 -11350.191,E2 -11350.191} C_VEL
LIN {X 0,Y 397.228,Z 424.622,A -85,B 0,C 180,E1 -11353.321,E2 -11353.321} C_VEL
LIN {X 0,Y 397.184,Z 424.634,A -85,B 0,C 180,E1 -11357.155,E2 -11357.155} C_VEL
LIN {X 0,Y 397.104,Z 424.647,A -85,B 0,C 180,E1 -11360.73,E2 -11360.73} C_VEL
LIN {X 0,Y 397.13,Z 424.64,A -85,B 0,C 180,E1 -11364.019,E2 -11364.019} C_VEL
LIN {X 0,Y 397.196,Z 424.632,A -85,B 0,C 180,E1 -11367.39,E2 -11367.39} C_VEL
LIN {X 0,Y 397.08,Z 424.647,A -85,B 0,C 180,E1 -11370.882,E2 -11370.882} C_VEL
LIN {X 0,Y 397.127,Z 424.645,A -85,B 0,C 180,E1 -11374.493,E2 -11374.493} C_VEL
LIN {X 0,Y 397.105,Z 424.646,A -85,B 0,C 180,E1 -11378.275,E2 -11378.275} C_VEL
LIN {X 0,Y 397.091,Z 424.65,A -85,B 0,C 180,E1 -11380.909,E2 -11380.909} C_VEL
LIN {X 0,Y 397.106,Z 424.648,A -85,B 0,C 180,E1 -11383.648,E2 -11383.648} C_VEL
LIN {X 0,Y 397.105,Z 424.665,A -85,B 0,C 180,E1 -11385.597,E2 -11385.597} C_VEL
LIN {X 0,Y 398.722,Z 432.777,A -85,B 0,C 180,E1 -11388.514,E2 -11388.514} C_VEL
LIN {X 0,Y 399.749,Z 439.022,A -85,B 0,C 180,E1 -11390.734,E2 -11390.734} C_VEL
LIN {X 0,Y 399.551,Z 445.017,A -85,B 0,C 180,E1 -11392.78,E2 -11392.78} C_VEL
LIN {X 0,Y 399.058,Z 455.6,A -85,B 0,C 180,E1 -11396.382,E2 -11396.382} C_VEL
LIN {X 0,Y 398.645,Z 465.599,A -85,B 0,C 180,E1 -11399.753,E2 -11399.753} C_VEL
LIN {X 0,Y 398.27,Z 474.489,A -85,B 0,C 180,E1 -11402.69,E2 -11402.69} C_VEL
LIN {X 0,Y 397.919,Z 484.905,A -85,B 0,C 180,E1 -11406.032,E2 -11406.032} C_VEL
LIN {X 0,Y 397.723,Z 491.221,A -85,B 0,C 180,E1 -11407.979,E2 -11407.979} C_VEL
LIN {X 0,Y 401.788,Z 508.365,A -85,B 0,C 180,E1 -11408.668,E2 -11408.668} C_VEL
LIN {X 0,Y 404.301,Z 522.503,A -85,B 0,C 180,E1 -11409.4,E2 -11409.4} C_VEL
LIN {X 0,Y 403.627,Z 536.037,A -85,B 0,C 180,E1 -11410.154,E2 -11410.154} C_VEL
LIN {X 0,Y 402.716,Z 548.349,A -85,B 0,C 180,E1 -11411.032,E2 -11411.032} C_VEL
LIN {X 0,Y 401.528,Z 561.007,A -85,B 0,C 180,E1 -11412.163,E2 -11412.163} C_VEL
LIN {X 0,Y 400.478,Z 571.388,A -85,B 0,C 180,E1 -11413.3,E2 -11413.3} C_VEL
LIN {X 0,Y 399.375,Z 581.924,A -85,B 0,C 180,E1 -11414.695,E2 -11414.695} C_VEL
LIN {X 0,Y 398.349,Z 591.229,A -85,B 0,C 180,E1 -11416.185,E2 -11416.185} C_VEL
LIN {X 0,Y 397.655,Z 599.313,A -85,B 0,C 180,E1 -11417.755,E2 -11417.755} C_VEL
LIN {X 0,Y 396.958,Z 605.875,A -85,B 0,C 180,E1 -11419.286,E2 -11419.286} C_VEL
LIN {X 0,Y 396.49,Z 611.322,A -85,B 0,C 180,E1 -11420.82,E2 -11420.82} C_VEL
LIN {X 0,Y 396.071,Z 617.026,A -85,B 0,C 180,E1 -11422.865,E2 -11422.865} C_VEL
LIN {X 0,Y 395.882,Z 621.175,A -85,B 0,C 180,E1 -11424.907,E2 -11424.907} C_VEL
LIN {X 0,Y 395.722,Z 623.894,A -85,B 0,C 180,E1 -11426.946,E2 -11426.946} C_VEL
LIN {X 0,Y 395.757,Z 625.257,A -85,B 0,C 180,E1 -11428.982,E2 -11428.982} C_VEL
LIN {X 0,Y 395.757,Z 625.294,A -85,B 0,C 180,E1 -11431.018,E2 -11431.018} C_VEL
LIN {X 0,Y 395.721,Z 623.994,A -85,B 0,C 180,E1 -11433.054,E2 -11433.054} C_VEL
LIN {X 0,Y 395.877,Z 621.335,A -85,B 0,C 180,E1 -11435.093,E2 -11435.093} C_VEL
LIN {X 0,Y 396.07,Z 617.252,A -85,B 0,C 180,E1 -11437.135,E2 -11437.135} C_VEL
LIN {X 0,Y 396.47,Z 611.617,A -85,B 0,C 180,E1 -11439.18,E2 -11439.18} C_VEL
LIN {X 0,Y 396.951,Z 605.686,A -85,B 0,C 180,E1 -11440.857,E2 -11440.857} C_VEL
LIN {X 0,Y 396.55,Z 602.77,A -85,B 0,C 180,E1 -11441.599,E2 -11441.599} C_VEL
LIN {X 0,Y 394.23,Z 597.799,A -85,B 0,C 180,E1 -11442.8,E2 -11442.8} C_VEL
LIN {X 0,Y 392.03,Z 592.31,A -85,B 0,C 180,E1 -11443.962,E2 -11443.962} C_VEL
LIN {X 0,Y 391.812,Z 588.581,A -85,B 0,C 180,E1 -11444.631,E2 -11444.631} C_VEL
LIN {X 0,Y 392.844,Z 579.088,A -85,B 0,C 180,E1 -11446.099,E2 -11446.099} C_VEL
LIN {X 0,Y 394.013,Z 567.886,A -85,B 0,C 180,E1 -11447.518,E2 -11447.518} C_VEL
LIN {X 0,Y 395.395,Z 555.374,A -85,B 0,C 180,E1 -11448.794,E2 -11448.794} C_VEL
LIN {X 0,Y 396.492,Z 542.992,A -85,B 0,C 180,E1 -11449.812,E2 -11449.812} C_VEL
LIN {X 0,Y 397.376,Z 530.713,A -85,B 0,C 180,E1 -11450.612,E2 -11450.612} C_VEL
LIN {X 0,Y 397.625,Z 523.886,A -85,B 0,C 180,E1 -11450.987,E2 -11450.987} C_VEL
LIN {X 0,Y 395.215,Z 509.668,A -85,B 0,C 180,E1 -11451.758,E2 -11451.758} C_VEL
LIN {X 0,Y 391.722,Z 495.266,A -85,B 0,C 180,E1 -11452.376,E2 -11452.376} C_VEL
LIN {X 0,Y 390.724,Z 491.199,A -85,B 0,C 180,E1 -11452.541,E2 -11452.541} C_VEL
LIN {X 0,Y 391.065,Z 481.639,A -85,B 0,C 180,E1 -11455.551,E2 -11455.551} C_VEL
LIN {X 0,Y 391.507,Z 471.139,A -85,B 0,C 180,E1 -11458.992,E2 -11458.992} C_VEL
LIN {X 0,Y 391.967,Z 460.545,A -85,B 0,C 180,E1 -11462.572,E2 -11462.572} C_VEL
LIN {X 0,Y 392.354,Z 451.754,A -85,B 0,C 180,E1 -11465.602,E2 -11465.602} C_VEL
LIN {X 0,Y 392.925,Z 442.546,A -85,B 0,C 180,E1 -11468.757,E2 -11468.757} C_VEL
LIN {X 0,Y 392.373,Z 437.283,A -85,B 0,C 180,E1 -11470.641,E2 -11470.641} C_VEL
LIN {X 0,Y 390.599,Z 428.174,A -85,B 0,C 180,E1 -11473.969,E2 -11473.969} C_VEL
LIN {X 0,Y 390.049,Z 425.525,A -85,B 0,C 180,E1 -11474.971,E2 -11474.971} C_VEL
LIN {X 0,Y 390.034,Z 425.53,A -85,B 0,C 180,E1 -11478.187,E2 -11478.187} C_VEL
LIN {X 0,Y 390.092,Z 425.521,A -85,B 0,C 180,E1 -11480.908,E2 -11480.908} C_VEL
LIN {X 0,Y 390.087,Z 425.521,A -85,B 0,C 180,E1 -11484.793,E2 -11484.793} C_VEL
LIN {X 0,Y 390.03,Z 425.527,A -85,B 0,C 180,E1 -11488.496,E2 -11488.496} C_VEL
LIN {X 0,Y 390.119,Z 425.516,A -85,B 0,C 180,E1 -11492.07,E2 -11492.07} C_VEL
LIN {X 0,Y 390.085,Z 425.519,A -85,B 0,C 180,E1 -11495.519,E2 -11495.519} C_VEL
LIN {X 0,Y 390.098,Z 425.517,A -85,B 0,C 180,E1 -11496.06,E2 -11496.06} C_VEL
LIN {X 0,Y 394.739,Z 439.694,A -85,B 0,C 180,E1 -11497.127,E2 -11497.127} C_VEL
LIN {X 0,Y 397.848,Z 449.613,A -85,B 0,C 180,E1 -11497.975,E2 -11497.975} C_VEL
LIN {X 0,Y 396.705,Z 463.865,A -85,B 0,C 180,E1 -11499.112,E2 -11499.112} C_VEL
LIN {X 0,Y 395.549,Z 476.481,A -85,B 0,C 180,E1 -11500.337,E2 -11500.337} C_VEL
LIN {X 0,Y 394.36,Z 489.164,A -85,B 0,C 180,E1 -11501.828,E2 -11501.828} C_VEL
LIN {X 0,Y 393.324,Z 500.226,A -85,B 0,C 180,E1 -11503.388,E2 -11503.388} C_VEL
LIN {X 0,Y 392.362,Z 509.589,A -85,B 0,C 180,E1 -11504.946,E2 -11504.946} C_VEL
LIN {X 0,Y 391.629,Z 517.522,A -85,B 0,C 180,E1 -11506.509,E2 -11506.509} C_VEL
LIN {X 0,Y 390.848,Z 525.309,A -85,B 0,C 180,E1 -11508.329,E2 -11508.329} C_VEL
LIN {X 0,Y 390.307,Z 531.717,A -85,B 0,C 180,E1 -11510.15,E2 -11510.15} C_VEL
LIN {X 0,Y 389.846,Z 537.718,A -85,B 0,C 180,E1 -11512.281,E2 -11512.281} C_VEL
LIN {X 0,Y 389.577,Z 541.1,A -85,B 0,C 180,E1 -11513.786,E2 -11513.786} C_VEL
LIN {X 0,Y 389.537,Z 544.564,A -85,B 0,C 180,E1 -11515.861,E2 -11515.861} C_VEL
LIN {X 0,Y 389.18,Z 546.808,A -85,B 0,C 180,E1 -11517.93,E2 -11517.93} C_VEL
LIN {X 0,Y 389.098,Z 547.838,A -85,B 0,C 180,E1 -11520,E2 -11520} C_VEL
LIN {X 0,Y 389.233,Z 547.679,A -85,B 0,C 180,E1 -11522.069,E2 -11522.069} C_VEL
LIN {X 0,Y 389.626,Z 546.321,A -85,B 0,C 180,E1 -11524.137,E2 -11524.137} C_VEL
LIN {X 0,Y 389.856,Z 545.193,A -85,B 0,C 180,E1 -11525.171,E2 -11525.171} C_VEL
LIN {X 0,Y 390.15,Z 542.035,A -85,B 0,C 180,E1 -11527.244,E2 -11527.244} C_VEL
LIN {X 0,Y 390.767,Z 537.521,A -85,B 0,C 180,E1 -11529.315,E2 -11529.315} C_VEL
LIN {X 0,Y 391.3,Z 531.615,A -85,B 0,C 180,E1 -11531.395,E2 -11531.395} C_VEL
LIN {X 0,Y 392.367,Z 524.021,A -85,B 0,C 180,E1 -11533.465,E2 -11533.465} C_VEL
LIN {X 0,Y 393.336,Z 516.562,A -85,B 0,C 180,E1 -11535.125,E2 -11535.125} C_VEL
LIN {X 0,Y 394.53,Z 507.411,A -85,B 0,C 180,E1 -11536.826,E2 -11536.826} C_VEL
LIN {X 0,Y 395.691,Z 497.459,A -85,B 0,C 180,E1 -11538.377,E2 -11538.377} C_VEL
LIN {X 0,Y 397.135,Z 485.451,A -85,B 0,C 180,E1 -11539.915,E2 -11539.915} C_VEL
LIN {X 0,Y 398.48,Z 473.418,A -85,B 0,C 180,E1 -11541.196,E2 -11541.196} C_VEL
LIN {X 0,Y 399.714,Z 460.322,A -85,B 0,C 180,E1 -11542.347,E2 -11542.347} C_VEL
LIN {X 0,Y 400.39,Z 451.458,A -85,B 0,C 180,E1 -11543.012,E2 -11543.012} C_VEL
LIN {X 0,Y 396.579,Z 440.364,A -85,B 0,C 180,E1 -11544.123,E2 -11544.123} C_VEL
LIN {X 0,Y 391.52,Z 428.962,A -85,B 0,C 180,E1 -11545.269,E2 -11545.269} C_VEL
LIN {X 0,Y 390.257,Z 426.257,A -85,B 0,C 180,E1 -11545.538,E2 -11545.538} C_VEL
LIN {X 0,Y 390.112,Z 425.521,A -85,B 0,C 180,E1 -11545.618,E2 -11545.618} C_VEL
LIN {X 0,Y 390.098,Z 425.522,A -85,B 0,C 180,E1 -11548.02,E2 -11548.02} C_VEL
LIN {X 0,Y 390.025,Z 425.53,A -85,B 0,C 180,E1 -11551.504,E2 -11551.504} C_VEL
LIN {X 0,Y 390.086,Z 425.522,A -85,B 0,C 180,E1 -11555.207,E2 -11555.207} C_VEL
LIN {X 0,Y 390.072,Z 425.524,A -85,B 0,C 180,E1 -11559.219,E2 -11559.219} C_VEL
LIN {X 0,Y 390.109,Z 425.728,A -85,B 0,C 180,E1 -11560.269,E2 -11560.269} C_VEL
LIN {X 0,Y 390.892,Z 430.098,A -85,B 0,C 180,E1 -11563.095,E2 -11563.095} C_VEL
LIN {X 0,Y 390.983,Z 432.618,A -85,B 0,C 180,E1 -11564.51,E2 -11564.51} C_VEL
LIN {X 0,Y 390.288,Z 440.116,A -85,B 0,C 180,E1 -11568.22,E2 -11568.22} C_VEL
LIN {X 0,Y 390.132,Z 447.535,A -85,B 0,C 180,E1 -11571.574,E2 -11571.574} C_VEL
LIN {X 0,Y 390.077,Z 455.114,A -85,B 0,C 180,E1 -11574.792,E2 -11574.792} C_VEL
LIN {X 0,Y 389.914,Z 464.226,A -85,B 0,C 180,E1 -11578.486,E2 -11578.486} C_VEL
LIN {X 0,Y 389.768,Z 473.257,A -85,B 0,C 180,E1 -11582.043,E2 -11582.043} C_VEL
LIN {X 0,Y 389.583,Z 482.133,A -85,B 0,C 180,E1 -11585.486,E2 -11585.486} C_VEL
LIN {X 0,Y 389.56,Z 484.203,A -85,B 0,C 180,E1 -11586.285,E2 -11586.285} C_VEL
LIN {X 0,Y 390.302,Z 488.114,A -85,B 0,C 180,E1 -11586.497,E2 -11586.497} C_VEL
LIN {X 0,Y 393.141,Z 502.39,A -85,B 0,C 180,E1 -11587.328,E2 -11587.328} C_VEL
LIN {X 0,Y 394.609,Z 517.223,A -85,B 0,C 180,E1 -11588.234,E2 -11588.234} C_VEL
LIN {X 0,Y 395.746,Z 528.183,A -85,B 0,C 180,E1 -11589.017,E2 -11589.017} C_VEL
LIN {X 0,Y 396.752,Z 536.012,A -85,B 0,C 180,E1 -11589.549,E2 -11589.549} C_VEL
LIN {X 0,Y 395.836,Z 549.667,A -85,B 0,C 180,E1 -11590.42,E2 -11590.42} C_VEL
LIN {X 0,Y 394.722,Z 562.218,A -85,B 0,C 180,E1 -11591.442,E2 -11591.442} C_VEL
LIN {X 0,Y 393.582,Z 573.642,A -85,B 0,C 180,E1 -11592.597,E2 -11592.597} C_VEL
LIN {X 0,Y 392.546,Z 584.107,A -85,B 0,C 180,E1 -11593.889,E2 -11593.889} C_VEL
LIN {X 0,Y 391.466,Z 594.488,A -85,B 0,C 180,E1 -11595.443,E2 -11595.443} C_VEL
LIN {X 0,Y 390.678,Z 603.028,A -85,B 0,C 180,E1 -11597.005,E2 -11597.005} C_VEL
LIN {X 0,Y 389.841,Z 611.159,A -85,B 0,C 180,E1 -11598.825,E2 -11598.825} C_VEL
LIN {X 0,Y 389.334,Z 617.69,A -85,B 0,C 180,E1 -11600.65,E2 -11600.65} C_VEL
LIN {X 0,Y 388.933,Z 623.461,A -85,B 0,C 180,E1 -11602.733,E2 -11602.733} C_VEL
LIN {X 0,Y 388.902,Z 625.744,A -85,B 0,C 180,E1 -11603.775,E2 -11603.775} C_VEL
LIN {X 0,Y 388.762,Z 629.192,A -85,B 0,C 180,E1 -11605.853,E2 -11605.853} C_VEL
LIN {X 0,Y 388.739,Z 631.234,A -85,B 0,C 180,E1 -11607.928,E2 -11607.928} C_VEL
LIN {X 0,Y 388.733,Z 631.913,A -85,B 0,C 180,E1 -11610,E2 -11610} C_VEL
LIN {X 0,Y 388.739,Z 631.234,A -85,B 0,C 180,E1 -11612.072,E2 -11612.072} C_VEL
LIN {X 0,Y 388.752,Z 629.194,A -85,B 0,C 180,E1 -11614.147,E2 -11614.147} C_VEL
LIN {X 0,Y 388.833,Z 625.743,A -85,B 0,C 180,E1 -11616.226,E2 -11616.226} C_VEL
LIN {X 0,Y 389.091,Z 620.777,A -85,B 0,C 180,E1 -11618.308,E2 -11618.308} C_VEL
LIN {X 0,Y 389.432,Z 615.958,A -85,B 0,C 180,E1 -11619.872,E2 -11619.872} C_VEL
LIN {X 0,Y 390.067,Z 608.982,A -85,B 0,C 180,E1 -11621.695,E2 -11621.695} C_VEL
LIN {X 0,Y 390.713,Z 601.667,A -85,B 0,C 180,E1 -11623.258,E2 -11623.258} C_VEL
LIN {X 0,Y 391.631,Z 592.85,A -85,B 0,C 180,E1 -11624.816,E2 -11624.816} C_VEL
LIN {X 0,Y 392.692,Z 582.141,A -85,B 0,C 180,E1 -11626.372,E2 -11626.372} C_VEL
LIN {X 0,Y 393.798,Z 571.276,A -85,B 0,C 180,E1 -11627.662,E2 -11627.662} C_VEL
LIN {X 0,Y 394.993,Z 559.349,A -85,B 0,C 180,E1 -11628.814,E2 -11628.814} C_VEL
LIN {X 0,Y 396.044,Z 546.893,A -85,B 0,C 180,E1 -11629.778,E2 -11629.778} C_VEL
LIN {X 0,Y 396.739,Z 534.597,A -85,B 0,C 180,E1 -11630.546,E2 -11630.546} C_VEL
LIN {X 0,Y 394.567,Z 520.265,A -85,B 0,C 180,E1 -11631.5,E2 -11631.5} C_VEL
LIN {X 0,Y 391.919,Z 505.312,A -85,B 0,C 180,E1 -11632.304,E2 -11632.304} C_VEL
LIN {X 0,Y 389.664,Z 493.884,A -85,B 0,C 180,E1 -11632.817,E2 -11632.817} C_VEL
LIN {X 0,Y 390.009,Z 486.161,A -85,B 0,C 180,E1 -11636.199,E2 -11636.199} C_VEL
LIN {X 0,Y 390.456,Z 478.37,A -85,B 0,C 180,E1 -11639.662,E2 -11639.662} C_VEL
LIN {X 0,Y 390.879,Z 470.447,A -85,B 0,C 180,E1 -11643.257,E2 -11643.257} C_VEL
LIN {X 0,Y 391.229,Z 463.776,A -85,B 0,C 180,E1 -11646.357,E2 -11646.357} C_VEL
LIN {X 0,Y 391.736,Z 455.662,A -85,B 0,C 180,E1 -11650.23,E2 -11650.23} C_VEL
LIN {X 0,Y 392.202,Z 448.882,A -85,B 0,C 180,E1 -11653.575,E2 -11653.575} C_VEL
LIN {X 0,Y 392.606,Z 443.227,A -85,B 0,C 180,E1 -11656.449,E2 -11656.449} C_VEL
LIN {X 0,Y 392.418,Z 438.822,A -85,B 0,C 180,E1 -11658.781,E2 -11658.781} C_VEL
LIN {X 0,Y 391.367,Z 432.812,A -85,B 0,C 180,E1 -11662.198,E2 -11662.198} C_VEL
LIN {X 0,Y 390.209,Z 426.35,A -85,B 0,C 180,E1 -11666.059,E2 -11666.059} C_VEL
LIN {X 0,Y 390.094,Z 425.519,A -85,B 0,C 180,E1 -11666.668,E2 -11666.668} C_VEL
LIN {X 0,Y 390.048,Z 425.528,A -85,B 0,C 180,E1 -11669.869,E2 -11669.869} C_VEL
LIN {X 0,Y 390.115,Z 425.506,A -85,B 0,C 180,E1 -11673.232,E2 -11673.232} C_VEL
LIN {X 0,Y 390.108,Z 425.517,A -85,B 0,C 180,E1 -11676.75,E2 -11676.75} C_VEL
LIN {X 0,Y 390.105,Z 425.505,A -85,B 0,C 180,E1 -11679.983,E2 -11679.983} C_VEL
LIN {X 0,Y 390.14,Z 425.512,A -85,B 0,C 180,E1 -11683.248,E2 -11683.248} C_VEL
LIN {X 0,Y 390.196,Z 425.5,A -85,B 0,C 180,E1 -11686.562,E2 -11686.562} C_VEL
LIN {X 0,Y 390.17,Z 425.503,A -85,B 0,C 180,E1 -11689.623,E2 -11689.623} C_VEL
LIN {X 0,Y 390.287,Z 425.492,A -85,B 0,C 180,E1 -11692.759,E2 -11692.759} C_VEL
LIN {X 0,Y 390.227,Z 425.501,A -85,B 0,C 180,E1 -11694.834,E2 -11694.834} C_VEL
LIN {X 0,Y 390.42,Z 425.468,A -85,B 0,C 180,E1 -11697.937,E2 -11697.937} C_VEL
LIN {X 0,Y 390.552,Z 425.464,A -85,B 0,C 180,E1 -11700,E2 -11700} C_VEL
LIN {X 0,Y 390.311,Z 425.479,A -85,B 0,C 180,E1 -11703.097,E2 -11703.097} C_VEL
LIN {X 0,Y 390.312,Z 425.488,A -85,B 0,C 180,E1 -11706.642,E2 -11706.642} C_VEL
LIN {X 0,Y 390.207,Z 425.496,A -85,B 0,C 180,E1 -11709.329,E2 -11709.329} C_VEL
LIN {X 0,Y 390.173,Z 425.505,A -85,B 0,C 180,E1 -11712.483,E2 -11712.483} C_VEL
LIN {X 0,Y 390.141,Z 425.513,A -85,B 0,C 180,E1 -11715.677,E2 -11715.677} C_VEL
LIN {X 0,Y 390.108,Z 425.508,A -85,B 0,C 180,E1 -11718.922,E2 -11718.922} C_VEL
LIN {X 0,Y 390.039,Z 425.522,A -85,B 0,C 180,E1 -11722.234,E2 -11722.234} C_VEL
LIN {X 0,Y 390.121,Z 425.513,A -85,B 0,C 180,E1 -11725.743,E2 -11725.743} C_VEL
LIN {X 0,Y 390.06,Z 425.522,A -85,B 0,C 180,E1 -11729.11,E2 -11729.11} C_VEL
LIN {X 0,Y 390.044,Z 425.523,A -85,B 0,C 180,E1 -11732.722,E2 -11732.722} C_VEL
LIN {X 0,Y 390.058,Z 425.52,A -85,B 0,C 180,E1 -11735.825,E2 -11735.825} C_VEL
LIN {X 0,Y 390.072,Z 425.523,A -85,B 0,C 180,E1 -11739.218,E2 -11739.218} C_VEL
LIN {X 0,Y 390.047,Z 425.528,A -85,B 0,C 180,E1 -11742.375,E2 -11742.375} C_VEL
LIN {X 0,Y 390.068,Z 425.608,A -85,B 0,C 180,E1 -11745.209,E2 -11745.209} C_VEL
LIN {X 0,Y 391.839,Z 434.391,A -85,B 0,C 180,E1 -11748.423,E2 -11748.423} C_VEL
LIN {X 0,Y 392.854,Z 440.941,A -85,B 0,C 180,E1 -11750.782,E2 -11750.782} C_VEL
LIN {X 0,Y 392.56,Z 447.781,A -85,B 0,C 180,E1 -11753.149,E2 -11753.149} C_VEL
LIN {X 0,Y 392.018,Z 458.584,A -85,B 0,C 180,E1 -11756.853,E2 -11756.853} C_VEL
LIN {X 0,Y 391.619,Z 469.088,A -85,B 0,C 180,E1 -11760.428,E2 -11760.428} C_VEL
LIN {X 0,Y 391.138,Z 479.759,A -85,B 0,C 180,E1 -11763.949,E2 -11763.949} C_VEL
LIN {X 0,Y 390.798,Z 490.208,A -85,B 0,C 180,E1 -11767.254,E2 -11767.254} C_VEL
LIN {X 0,Y 390.801,Z 491.433,A -85,B 0,C 180,E1 -11767.591,E2 -11767.591} C_VEL
LIN {X 0,Y 394.582,Z 506.809,A -85,B 0,C 180,E1 -11768.208,E2 -11768.208} C_VEL
LIN {X 0,Y 397.129,Z 520.424,A -85,B 0,C 180,E1 -11768.909,E2 -11768.909} C_VEL
LIN {X 0,Y 397.626,Z 525.801,A -85,B 0,C 180,E1 -11769.215,E2 -11769.215} C_VEL
LIN {X 0,Y 396.731,Z 539.384,A -85,B 0,C 180,E1 -11770.027,E2 -11770.027} C_VEL
LIN {X 0,Y 395.717,Z 551.471,A -85,B 0,C 180,E1 -11770.953,E2 -11770.953} C_VEL
LIN {X 0,Y 394.482,Z 563.578,A -85,B 0,C 180,E1 -11772.102,E2 -11772.102} C_VEL
LIN {X 0,Y 393.319,Z 574.566,A -85,B 0,C 180,E1 -11773.388,E2 -11773.388} C_VEL
LIN {X 0,Y 392.119,Z 585.361,A -85,B 0,C 180,E1 -11774.937,E2 -11774.937} C_VEL
LIN {X 0,Y 391.201,Z 594.277,A -85,B 0,C 180,E1 -11776.494,E2 -11776.494} C_VEL
LIN {X 0,Y 390.409,Z 601.704,A -85,B 0,C 180,E1 -11778.052,E2 -11778.052} C_VEL
LIN {X 0,Y 389.801,Z 607.894,A -85,B 0,C 180,E1 -11779.613,E2 -11779.613} C_VEL
LIN {X 0,Y 389.195,Z 614.436,A -85,B 0,C 180,E1 -11781.694,E2 -11781.694} C_VEL
LIN {X 0,Y 388.923,Z 619.345,A -85,B 0,C 180,E1 -11783.776,E2 -11783.776} C_VEL
LIN {X 0,Y 388.706,Z 622.766,A -85,B 0,C 180,E1 -11785.853,E2 -11785.853} C_VEL
LIN {X 0,Y 388.654,Z 624.8,A -85,B 0,C 180,E1 -11787.927,E2 -11787.927} C_VEL
LIN {X 0,Y 388.672,Z 625.501,A -85,B 0,C 180,E1 -11790,E2 -11790} C_VEL
LIN {X 0,Y 388.653,Z 624.87,A -85,B 0,C 180,E1 -11792.073,E2 -11792.073} C_VEL
LIN {X 0,Y 388.706,Z 622.894,A -85,B 0,C 180,E1 -11794.147,E2 -11794.147} C_VEL
LIN {X 0,Y 388.873,Z 619.429,A -85,B 0,C 180,E1 -11796.278,E2 -11796.278} C_VEL
LIN {X 0,Y 389.19,Z 614.694,A -85,B 0,C 180,E1 -11798.306,E2 -11798.306} C_VEL
LIN {X 0,Y 389.742,Z 608.22,A -85,B 0,C 180,E1 -11800.389,E2 -11800.389} C_VEL
LIN {X 0,Y 390.518,Z 601.003,A -85,B 0,C 180,E1 -11802.208,E2 -11802.208} C_VEL
LIN {X 0,Y 391.392,Z 592.284,A -85,B 0,C 180,E1 -11803.98,E2 -11803.98} C_VEL
LIN {X 0,Y 391.812,Z 588.581,A -85,B 0,C 180,E1 -11804.631,E2 -11804.631} C_VEL
LIN {X 0,Y 391.617,Z 584.742,A -85,B 0,C 180,E1 -11805.283,E2 -11805.283} C_VEL
LIN {X 0,Y 389.57,Z 578.307,A -85,B 0,C 180,E1 -11806.353,E2 -11806.353} C_VEL
LIN {X 0,Y 387.523,Z 571.516,A -85,B 0,C 180,E1 -11807.374,E2 -11807.374} C_VEL
LIN {X 0,Y 387.323,Z 567.013,A -85,B 0,C 180,E1 -11807.939,E2 -11807.939} C_VEL
LIN {X 0,Y 388.667,Z 555.412,A -85,B 0,C 180,E1 -11809.132,E2 -11809.132} C_VEL
LIN {X 0,Y 389.807,Z 543.023,A -85,B 0,C 180,E1 -11810.166,E2 -11810.166} C_VEL
LIN {X 0,Y 390.807,Z 529.084,A -85,B 0,C 180,E1 -11811.08,E2 -11811.08} C_VEL
LIN {X 0,Y 390.862,Z 524.4,A -85,B 0,C 180,E1 -11811.34,E2 -11811.34} C_VEL
LIN {X 0,Y 388.608,Z 511.171,A -85,B 0,C 180,E1 -11812.086,E2 -11812.086} C_VEL
LIN {X 0,Y 385.345,Z 497.313,A -85,B 0,C 180,E1 -11812.717,E2 -11812.717} C_VEL
LIN {X 0,Y 383.801,Z 491.194,A -85,B 0,C 180,E1 -11812.971,E2 -11812.971} C_VEL
LIN {X 0,Y 384.232,Z 479.551,A -85,B 0,C 180,E1 -11816.692,E2 -11816.692} C_VEL
LIN {X 0,Y 384.692,Z 469.197,A -85,B 0,C 180,E1 -11820.159,E2 -11820.159} C_VEL
LIN {X 0,Y 385.2,Z 458.574,A -85,B 0,C 180,E1 -11823.812,E2 -11823.812} C_VEL
LIN {X 0,Y 385.782,Z 447.625,A -85,B 0,C 180,E1 -11827.61,E2 -11827.61} C_VEL
LIN {X 0,Y 385.912,Z 441.971,A -85,B 0,C 180,E1 -11829.598,E2 -11829.598} C_VEL
LIN {X 0,Y 384.749,Z 435.112,A -85,B 0,C 180,E1 -11832.132,E2 -11832.132} C_VEL
LIN {X 0,Y 383.025,Z 426.403,A -85,B 0,C 180,E1 -11835.419,E2 -11835.419} C_VEL
LIN {X 0,Y 382.99,Z 426.409,A -85,B 0,C 180,E1 -11838.796,E2 -11838.796} C_VEL
LIN {X 0,Y 383.003,Z 426.406,A -85,B 0,C 180,E1 -11842.096,E2 -11842.096} C_VEL
LIN {X 0,Y 383.02,Z 426.396,A -85,B 0,C 180,E1 -11845.332,E2 -11845.332} C_VEL
LIN {X 0,Y 382.988,Z 426.396,A -85,B 0,C 180,E1 -11849.082,E2 -11849.082} C_VEL
LIN {X 0,Y 383.058,Z 426.397,A -85,B 0,C 180,E1 -11852.698,E2 -11852.698} C_VEL
LIN {X 0,Y 383.064,Z 426.393,A -85,B 0,C 180,E1 -11855.715,E2 -11855.715} C_VEL
LIN {X 0,Y 388.442,Z 442.843,A -85,B 0,C 180,E1 -11856.995,E2 -11856.995} C_VEL
LIN {X 0,Y 390.831,Z 450.458,A -85,B 0,C 180,E1 -11857.674,E2 -11857.674} C_VEL
LIN {X 0,Y 390.696,Z 455.646,A -85,B 0,C 180,E1 -11858.083,E2 -11858.083} C_VEL
LIN {X 0,Y 389.515,Z 469.173,A -85,B 0,C 180,E1 -11859.262,E2 -11859.262} C_VEL
LIN {X 0,Y 388.334,Z 481.737,A -85,B 0,C 180,E1 -11860.591,E2 -11860.591} C_VEL
LIN {X 0,Y 387.195,Z 493.1,A -85,B 0,C 180,E1 -11862.027,E2 -11862.027} C_VEL
LIN {X 0,Y 386.114,Z 503.66,A -85,B 0,C 180,E1 -11863.613,E2 -11863.613} C_VEL
LIN {X 0,Y 384.998,Z 513.411,A -85,B 0,C 180,E1 -11865.352,E2 -11865.352} C_VEL
LIN {X 0,Y 384.384,Z 521.368,A -85,B 0,C 180,E1 -11867.057,E2 -11867.057} C_VEL
LIN {X 0,Y 383.61,Z 528.642,A -85,B 0,C 180,E1 -11868.909,E2 -11868.909} C_VEL
LIN {X 0,Y 383.057,Z 535.353,A -85,B 0,C 180,E1 -11871.028,E2 -11871.028} C_VEL
LIN {X 0,Y 382.644,Z 540.285,A -85,B 0,C 180,E1 -11873.007,E2 -11873.007} C_VEL
LIN {X 0,Y 382.526,Z 543.626,A -85,B 0,C 180,E1 -11874.729,E2 -11874.729} C_VEL
LIN {X 0,Y 382.328,Z 546.525,A -85,B 0,C 180,E1 -11876.839,E2 -11876.839} C_VEL
LIN {X 0,Y 382.039,Z 548.227,A -85,B 0,C 180,E1 -11878.946,E2 -11878.946} C_VEL
LIN {X 0,Y 382.081,Z 548.724,A -85,B 0,C 180,E1 -11881.054,E2 -11881.054} C_VEL
LIN {X 0,Y 382.347,Z 548.023,A -85,B 0,C 180,E1 -11883.161,E2 -11883.161} C_VEL
LIN {X 0,Y 382.846,Z 546.111,A -85,B 0,C 180,E1 -11885.266,E2 -11885.266} C_VEL
LIN {X 0,Y 383.186,Z 543.008,A -85,B 0,C 180,E1 -11887.376,E2 -11887.376} C_VEL
LIN {X 0,Y 383.83,Z 538.569,A -85,B 0,C 180,E1 -11889.485,E2 -11889.485} C_VEL
LIN {X 0,Y 384.415,Z 532.708,A -85,B 0,C 180,E1 -11891.602,E2 -11891.602} C_VEL
LIN {X 0,Y 385.561,Z 525.166,A -85,B 0,C 180,E1 -11893.707,E2 -11893.707} C_VEL
LIN {X 0,Y 386.468,Z 518.694,A -85,B 0,C 180,E1 -11895.215,E2 -11895.215} C_VEL
LIN {X 0,Y 387.673,Z 510.257,A -85,B 0,C 180,E1 -11896.861,E2 -11896.861} C_VEL
LIN {X 0,Y 388.866,Z 500.656,A -85,B 0,C 180,E1 -11898.438,E2 -11898.438} C_VEL
LIN {X 0,Y 390.347,Z 489.227,A -85,B 0,C 180,E1 -11900.004,E2 -11900.004} C_VEL
LIN {X 0,Y 391.824,Z 477.743,A -85,B 0,C 180,E1 -11901.298,E2 -11901.298} C_VEL
LIN {X 0,Y 393.212,Z 463.868,A -85,B 0,C 180,E1 -11902.599,E2 -11902.599} C_VEL
LIN {X 0,Y 394.112,Z 453.66,A -85,B 0,C 180,E1 -11903.4,E2 -11903.4} C_VEL
LIN {X 0,Y 390.285,Z 442.497,A -85,B 0,C 180,E1 -11904.58,E2 -11904.58} C_VEL
LIN {X 0,Y 384.575,Z 429.933,A -85,B 0,C 180,E1 -11905.941,E2 -11905.941} C_VEL
LIN {X 0,Y 383.232,Z 427.292,A -85,B 0,C 180,E1 -11906.233,E2 -11906.233} C_VEL
LIN {X 0,Y 383.073,Z 426.399,A -85,B 0,C 180,E1 -11906.315,E2 -11906.315} C_VEL
LIN {X 0,Y 382.993,Z 426.407,A -85,B 0,C 180,E1 -11909.7,E2 -11909.7} C_VEL
LIN {X 0,Y 383.004,Z 426.403,A -85,B 0,C 180,E1 -11913.401,E2 -11913.401} C_VEL
LIN {X 0,Y 383.033,Z 426.399,A -85,B 0,C 180,E1 -11916.165,E2 -11916.165} C_VEL
LIN {X 0,Y 383.079,Z 426.524,A -85,B 0,C 180,E1 -11919.723,E2 -11919.723} C_VEL
LIN {X 0,Y 383.904,Z 431.246,A -85,B 0,C 180,E1 -11922.923,E2 -11922.923} C_VEL
LIN {X 0,Y 384.022,Z 433.893,A -85,B 0,C 180,E1 -11924.46,E2 -11924.46} C_VEL
LIN {X 0,Y 383.286,Z 440.81,A -85,B 0,C 180,E1 -11927.989,E2 -11927.989} C_VEL
LIN {X 0,Y 383.146,Z 447.018,A -85,B 0,C 180,E1 -11930.905,E2 -11930.905} C_VEL
LIN {X 0,Y 383.021,Z 455.655,A -85,B 0,C 180,E1 -11934.691,E2 -11934.691} C_VEL
LIN {X 0,Y 382.844,Z 464.704,A -85,B 0,C 180,E1 -11938.454,E2 -11938.454} C_VEL
LIN {X 0,Y 382.714,Z 473.041,A -85,B 0,C 180,E1 -11941.818,E2 -11941.818} C_VEL
LIN {X 0,Y 382.488,Z 482.533,A -85,B 0,C 180,E1 -11945.58,E2 -11945.58} C_VEL
LIN {X 0,Y 383.236,Z 486.38,A -85,B 0,C 180,E1 -11945.804,E2 -11945.804} C_VEL
LIN {X 0,Y 386.058,Z 499.45,A -85,B 0,C 180,E1 -11946.627,E2 -11946.627} C_VEL
LIN {X 0,Y 387.694,Z 512.772,A -85,B 0,C 180,E1 -11947.482,E2 -11947.482} C_VEL
LIN {X 0,Y 388.758,Z 527.331,A -85,B 0,C 180,E1 -11948.527,E2 -11948.527} C_VEL
LIN {X 0,Y 389.843,Z 534.751,A -85,B 0,C 180,E1 -11949.094,E2 -11949.094} C_VEL
LIN {X 0,Y 389.946,Z 538.463,A -85,B 0,C 180,E1 -11949.327,E2 -11949.327} C_VEL
LIN {X 0,Y 388.967,Z 551.667,A -85,B 0,C 180,E1 -11950.219,E2 -11950.219} C_VEL
LIN {X 0,Y 387.87,Z 563.6,A -85,B 0,C 180,E1 -11951.239,E2 -11951.239} C_VEL
LIN {X 0,Y 386.675,Z 574.769,A -85,B 0,C 180,E1 -11952.412,E2 -11952.412} C_VEL
LIN {X 0,Y 385.508,Z 585.95,A -85,B 0,C 180,E1 -11953.858,E2 -11953.858} C_VEL
LIN {X 0,Y 384.375,Z 596.244,A -85,B 0,C 180,E1 -11955.494,E2 -11955.494} C_VEL
LIN {X 0,Y 383.489,Z 605.45,A -85,B 0,C 180,E1 -11957.296,E2 -11957.296} C_VEL
LIN {X 0,Y 382.739,Z 612.112,A -85,B 0,C 180,E1 -11958.883,E2 -11958.883} C_VEL
LIN {X 0,Y 382.306,Z 617.634,A -85,B 0,C 180,E1 -11960.477,E2 -11960.477} C_VEL
LIN {X 0,Y 381.86,Z 623.404,A -85,B 0,C 180,E1 -11962.598,E2 -11962.598} C_VEL
LIN {X 0,Y 381.809,Z 625.794,A -85,B 0,C 180,E1 -11963.712,E2 -11963.712} C_VEL
LIN {X 0,Y 381.684,Z 629.135,A -85,B 0,C 180,E1 -11965.776,E2 -11965.776} C_VEL
LIN {X 0,Y 381.634,Z 631.175,A -85,B 0,C 180,E1 -11967.889,E2 -11967.889} C_VEL
LIN {X 0,Y 381.645,Z 631.855,A -85,B 0,C 180,E1 -11970,E2 -11970} C_VEL
LIN {X 0,Y 381.634,Z 631.176,A -85,B 0,C 180,E1 -11972.111,E2 -11972.111} C_VEL
LIN {X 0,Y 381.672,Z 629.136,A -85,B 0,C 180,E1 -11974.224,E2 -11974.224} C_VEL
LIN {X 0,Y 381.766,Z 625.685,A -85,B 0,C 180,E1 -11976.342,E2 -11976.342} C_VEL
LIN {X 0,Y 382.024,Z 620.719,A -85,B 0,C 180,E1 -11978.463,E2 -11978.463} C_VEL
LIN {X 0,Y 382.394,Z 615.9,A -85,B 0,C 180,E1 -11980.055,E2 -11980.055} C_VEL
LIN {X 0,Y 383.09,Z 608.926,A -85,B 0,C 180,E1 -11981.911,E2 -11981.911} C_VEL
LIN {X 0,Y 383.907,Z 600.258,A -85,B 0,C 180,E1 -11983.768,E2 -11983.768} C_VEL
LIN {X 0,Y 384.873,Z 591.17,A -85,B 0,C 180,E1 -11985.354,E2 -11985.354} C_VEL
LIN {X 0,Y 386.04,Z 580.116,A -85,B 0,C 180,E1 -11986.935,E2 -11986.935} C_VEL
LIN {X 0,Y 387.33,Z 568.789,A -85,B 0,C 180,E1 -11988.24,E2 -11988.24} C_VEL
LIN {X 0,Y 388.547,Z 556.482,A -85,B 0,C 180,E1 -11989.39,E2 -11989.39} C_VEL
